LIN {X 0,Y 523.368,Z 555.346,A -85,B 0,C 180,E1 -4773.08,E2 -4773.08} C_VEL
LIN {X 0,Y 523.424,Z 552.407,A -85,B 0,C 180,E1 -4774.236,E2 -4774.236} C_VEL
LIN {X 0,Y 523.462,Z 548.426,A -85,B 0,C 180,E1 -4775.394,E2 -4775.394} C_VEL
LIN {X 0,Y 523.515,Z 542.323,A -85,B 0,C 180,E1 -4776.743,E2 -4776.743} C_VEL
LIN {X 0,Y 523.667,Z 535.613,A -85,B 0,C 180,E1 -4777.908,E2 -4777.908} C_VEL
LIN {X 0,Y 523.85,Z 527.313,A -85,B 0,C 180,E1 -4779.071,E2 -4779.071} C_VEL
LIN {X 0,Y 524.066,Z 518.806,A -85,B 0,C 180,E1 -4780.041,E2 -4780.041} C_VEL
LIN {X 0,Y 524.361,Z 508.295,A -85,B 0,C 180,E1 -4781.012,E2 -4781.012} C_VEL
LIN {X 0,Y 524.634,Z 497.983,A -85,B 0,C 180,E1 -4781.783,E2 -4781.783} C_VEL
LIN {X 0,Y 524.903,Z 486.499,A -85,B 0,C 180,E1 -4782.469,E2 -4782.469} C_VEL
LIN {X 0,Y 525.115,Z 474.788,A -85,B 0,C 180,E1 -4783.005,E2 -4783.005} C_VEL
LIN {X 0,Y 525.386,Z 461.299,A -85,B 0,C 180,E1 -4783.441,E2 -4783.441} C_VEL
LIN {X 0,Y 525.56,Z 447.895,A -85,B 0,C 180,E1 -4783.707,E2 -4783.707} C_VEL
LIN {X 0,Y 525.818,Z 355.734,A -85,B 0,C 180,E1 -4784.974,E2 -4784.974} C_VEL
LIN {X 0,Y 524.289,Z 345.618,A -85,B 0,C 180,E1 -4785.171,E2 -4785.171} C_VEL
LIN {X 0,Y 524.744,Z 323.595,A -85,B 0,C 180,E1 -4788.528,E2 -4788.528} C_VEL
LIN {X 0,Y 525.163,Z 305.11,A -85,B 0,C 180,E1 -4791.388,E2 -4791.388} C_VEL
LIN {X 0,Y 525.41,Z 293.296,A -85,B 0,C 180,E1 -4793.242,E2 -4793.242} C_VEL
LIN {X 0,Y 523.995,Z 285.213,A -85,B 0,C 180,E1 -4794.622,E2 -4794.622} C_VEL
LIN {X 0,Y 523.978,Z 285.217,A -85,B 0,C 180,E1 -4797.718,E2 -4797.718} C_VEL
LIN {X 0,Y 523.951,Z 285.214,A -85,B 0,C 180,E1 -4800.855,E2 -4800.855} C_VEL
LIN {X 0,Y 523.937,Z 285.217,A -85,B 0,C 180,E1 -4803.73,E2 -4803.73} C_VEL
LIN {X 0,Y 523.909,Z 285.228,A -85,B 0,C 180,E1 -4806.402,E2 -4806.402} C_VEL
LIN {X 0,Y 523.919,Z 285.218,A -85,B 0,C 180,E1 -4809.086,E2 -4809.086} C_VEL
LIN {X 0,Y 523.957,Z 285.216,A -85,B 0,C 180,E1 -4812.119,E2 -4812.119} C_VEL
LIN {X 0,Y 523.948,Z 285.215,A -85,B 0,C 180,E1 -4815.311,E2 -4815.311} C_VEL
LIN {X 0,Y 523.961,Z 285.221,A -85,B 0,C 180,E1 -4818.69,E2 -4818.69} C_VEL
LIN {X 0,Y 523.922,Z 285.223,A -85,B 0,C 180,E1 -4821.081,E2 -4821.081} C_VEL
LIN {X 0,Y 523.905,Z 285.219,A -85,B 0,C 180,E1 -4823.825,E2 -4823.825} C_VEL
LIN {X 0,Y 523.918,Z 285.221,A -85,B 0,C 180,E1 -4826.634,E2 -4826.634} C_VEL
LIN {X 0,Y 523.961,Z 285.218,A -85,B 0,C 180,E1 -4829.356,E2 -4829.356} C_VEL
LIN {X 0,Y 523.981,Z 285.209,A -85,B 0,C 180,E1 -4832.282,E2 -4832.282} C_VEL
LIN {X 0,Y 523.954,Z 285.214,A -85,B 0,C 180,E1 -4834.581,E2 -4834.581} C_VEL
LIN {X 0,Y 523.915,Z 285.224,A -85,B 0,C 180,E1 -4837.106,E2 -4837.106} C_VEL
LIN {X 0,Y 523.984,Z 285.212,A -85,B 0,C 180,E1 -4839.866,E2 -4839.866} C_VEL
LIN {X 0,Y 523.959,Z 285.213,A -85,B 0,C 180,E1 -4842.837,E2 -4842.837} C_VEL
LIN {X 0,Y 523.982,Z 285.213,A -85,B 0,C 180,E1 -4845.236,E2 -4845.236} C_VEL
LIN {X 0,Y 524.018,Z 285.206,A -85,B 0,C 180,E1 -4848.394,E2 -4848.394} C_VEL
LIN {X 0,Y 524.001,Z 285.212,A -85,B 0,C 180,E1 -4851.516,E2 -4851.516} C_VEL
LIN {X 0,Y 524.079,Z 285.198,A -85,B 0,C 180,E1 -4854.613,E2 -4854.613} C_VEL
LIN {X 0,Y 524.116,Z 285.197,A -85,B 0,C 180,E1 -4857.694,E2 -4857.694} C_VEL
LIN {X 0,Y 524.126,Z 285.193,A -85,B 0,C 180,E1 -4860.768,E2 -4860.768} C_VEL
LIN {X 0,Y 524.073,Z 285.198,A -85,B 0,C 180,E1 -4863.075,E2 -4863.075} C_VEL
LIN {X 0,Y 524.039,Z 285.21,A -85,B 0,C 180,E1 -4866.159,E2 -4866.159} C_VEL
LIN {X 0,Y 523.99,Z 285.208,A -85,B 0,C 180,E1 -4869.262,E2 -4869.262} C_VEL
LIN {X 0,Y 524.004,Z 285.207,A -85,B 0,C 180,E1 -4871.737,E2 -4871.737} C_VEL
LIN {X 0,Y 523.999,Z 285.21,A -85,B 0,C 180,E1 -4875.052,E2 -4875.052} C_VEL
LIN {X 0,Y 523.952,Z 285.214,A -85,B 0,C 180,E1 -4877.969,E2 -4877.969} C_VEL
LIN {X 0,Y 523.976,Z 285.214,A -85,B 0,C 180,E1 -4880.41,E2 -4880.41} C_VEL
LIN {X 0,Y 523.914,Z 285.228,A -85,B 0,C 180,E1 -4882.893,E2 -4882.893} C_VEL
LIN {X 0,Y 523.957,Z 285.215,A -85,B 0,C 180,E1 -4885.418,E2 -4885.418} C_VEL
LIN {X 0,Y 523.972,Z 285.21,A -85,B 0,C 180,E1 -4887.999,E2 -4887.999} C_VEL
LIN {X 0,Y 523.949,Z 285.219,A -85,B 0,C 180,E1 -4890.854,E2 -4890.854} C_VEL
LIN {X 0,Y 523.963,Z 285.214,A -85,B 0,C 180,E1 -4893.734,E2 -4893.734} C_VEL
LIN {X 0,Y 523.902,Z 285.219,A -85,B 0,C 180,E1 -4896.4,E2 -4896.4} C_VEL
LIN {X 0,Y 523.922,Z 285.222,A -85,B 0,C 180,E1 -4899.084,E2 -4899.084} C_VEL
LIN {X 0,Y 523.955,Z 285.214,A -85,B 0,C 180,E1 -4902.118,E2 -4902.118} C_VEL
LIN {X 0,Y 523.946,Z 285.219,A -85,B 0,C 180,E1 -4905.31,E2 -4905.31} C_VEL
LIN {X 0,Y 523.918,Z 285.218,A -85,B 0,C 180,E1 -4906.904,E2 -4906.904} C_VEL
LIN {X 0,Y 523.254,Z 285.308,A -85,B 0,C 180,E1 -4907.546,E2 -4907.546} C_VEL
LIN {X 0,Y 520.414,Z 285.662,A -85,B 0,C 180,E1 -4908.588,E2 -4908.588} C_VEL
LIN {X 0,Y 518.01,Z 285.961,A -85,B 0,C 180,E1 -4909.426,E2 -4909.426} C_VEL
LIN {X 0,Y 516.972,Z 286.088,A -85,B 0,C 180,E1 -4910.074,E2 -4910.074} C_VEL
LIN {X 0,Y 516.885,Z 286.096,A -85,B 0,C 180,E1 -4910.293,E2 -4910.293} C_VEL
LIN {X 0,Y 516.88,Z 286.096,A -85,B 0,C 180,E1 -4913.342,E2 -4913.342} C_VEL
LIN {X 0,Y 516.911,Z 286.097,A -85,B 0,C 180,E1 -4916.12,E2 -4916.12} C_VEL
LIN {X 0,Y 516.895,Z 286.092,A -85,B 0,C 180,E1 -4918.935,E2 -4918.935} C_VEL
LIN {X 0,Y 516.923,Z 286.091,A -85,B 0,C 180,E1 -4921.584,E2 -4921.584} C_VEL
LIN {X 0,Y 516.933,Z 286.098,A -85,B 0,C 180,E1 -4924.21,E2 -4924.21} C_VEL
LIN {X 0,Y 516.864,Z 286.099,A -85,B 0,C 180,E1 -4926.775,E2 -4926.775} C_VEL
LIN {X 0,Y 516.943,Z 286.087,A -85,B 0,C 180,E1 -4929.731,E2 -4929.731} C_VEL
LIN {X 0,Y 516.923,Z 286.097,A -85,B 0,C 180,E1 -4932.595,E2 -4932.595} C_VEL
LIN {X 0,Y 516.945,Z 286.089,A -85,B 0,C 180,E1 -4935.029,E2 -4935.029} C_VEL
LIN {X 0,Y 516.968,Z 286.086,A -85,B 0,C 180,E1 -4938.233,E2 -4938.233} C_VEL
LIN {X 0,Y 516.958,Z 286.088,A -85,B 0,C 180,E1 -4941.398,E2 -4941.398} C_VEL
LIN {X 0,Y 517.003,Z 286.083,A -85,B 0,C 180,E1 -4943.756,E2 -4943.756} C_VEL
LIN {X 0,Y 516.949,Z 286.257,A -85,B 0,C 180,E1 -4945.271,E2 -4945.271} C_VEL
LIN {X 0,Y 517.481,Z 291.535,A -85,B 0,C 180,E1 -4946.3,E2 -4946.3} C_VEL
LIN {X 0,Y 517.248,Z 305.925,A -85,B 0,C 180,E1 -4949.026,E2 -4949.026} C_VEL
LIN {X 0,Y 517.231,Z 309.396,A -85,B 0,C 180,E1 -4949.683,E2 -4949.683} C_VEL
LIN {X 0,Y 519.124,Z 320.066,A -85,B 0,C 180,E1 -4949.902,E2 -4949.902} C_VEL
LIN {X 0,Y 518.55,Z 416.495,A -85,B 0,C 180,E1 -4951.261,E2 -4951.261} C_VEL
LIN {X 0,Y 518.369,Z 430.247,A -85,B 0,C 180,E1 -4951.625,E2 -4951.625} C_VEL
LIN {X 0,Y 518.189,Z 442.011,A -85,B 0,C 180,E1 -4952.088,E2 -4952.088} C_VEL
LIN {X 0,Y 517.935,Z 453.991,A -85,B 0,C 180,E1 -4952.721,E2 -4952.721} C_VEL
LIN {X 0,Y 517.571,Z 465.423,A -85,B 0,C 180,E1 -4953.502,E2 -4953.502} C_VEL
LIN {X 0,Y 517.287,Z 475.712,A -85,B 0,C 180,E1 -4954.382,E2 -4954.382} C_VEL
LIN {X 0,Y 517.045,Z 484.149,A -85,B 0,C 180,E1 -4955.263,E2 -4955.263} C_VEL
LIN {X 0,Y 516.815,Z 491.954,A -85,B 0,C 180,E1 -4956.244,E2 -4956.244} C_VEL
LIN {X 0,Y 516.665,Z 499.581,A -85,B 0,C 180,E1 -4957.424,E2 -4957.424} C_VEL
LIN {X 0,Y 516.486,Z 505.737,A -85,B 0,C 180,E1 -4958.607,E2 -4958.607} C_VEL
LIN {X 0,Y 516.369,Z 510.631,A -85,B 0,C 180,E1 -4959.794,E2 -4959.794} C_VEL
LIN {X 0,Y 516.337,Z 514.4,A -85,B 0,C 180,E1 -4960.984,E2 -4960.984} C_VEL
LIN {X 0,Y 516.28,Z 516.352,A -85,B 0,C 180,E1 -4961.781,E2 -4961.781} C_VEL
LIN {X 0,Y 516.22,Z 517.869,A -85,B 0,C 180,E1 -4962.58,E2 -4962.58} C_VEL
LIN {X 0,Y 516.183,Z 518.924,A -85,B 0,C 180,E1 -4963.382,E2 -4963.382} C_VEL
LIN {X 0,Y 516.246,Z 519.808,A -85,B 0,C 180,E1 -4964.857,E2 -4964.857} C_VEL
LIN {X 0,Y 516.15,Z 519.646,A -85,B 0,C 180,E1 -4965.801,E2 -4965.801} C_VEL
LIN {X 0,Y 516.166,Z 519.025,A -85,B 0,C 180,E1 -4966.613,E2 -4966.613} C_VEL
LIN {X 0,Y 516.228,Z 517.656,A -85,B 0,C 180,E1 -4967.638,E2 -4967.638} C_VEL
LIN {X 0,Y 516.287,Z 514.52,A -85,B 0,C 180,E1 -4969.067,E2 -4969.067} C_VEL
LIN {X 0,Y 516.396,Z 510.398,A -85,B 0,C 180,E1 -4970.366,E2 -4970.366} C_VEL
LIN {X 0,Y 516.45,Z 505.433,A -85,B 0,C 180,E1 -4971.555,E2 -4971.555} C_VEL
LIN {X 0,Y 516.657,Z 498.795,A -85,B 0,C 180,E1 -4972.809,E2 -4972.809} C_VEL
LIN {X 0,Y 516.901,Z 490.288,A -85,B 0,C 180,E1 -4974.071,E2 -4974.071} C_VEL
LIN {X 0,Y 517.154,Z 481.46,A -85,B 0,C 180,E1 -4975.129,E2 -4975.129} C_VEL
LIN {X 0,Y 517.471,Z 471.556,A -85,B 0,C 180,E1 -4976.09,E2 -4976.09} C_VEL
LIN {X 0,Y 517.711,Z 460.662,A -85,B 0,C 180,E1 -4976.939,E2 -4976.939} C_VEL
LIN {X 0,Y 518.074,Z 448.787,A -85,B 0,C 180,E1 -4977.668,E2 -4977.668} C_VEL
LIN {X 0,Y 518.317,Z 437.639,A -85,B 0,C 180,E1 -4978.194,E2 -4978.194} C_VEL
LIN {X 0,Y 518.525,Z 425.119,A -85,B 0,C 180,E1 -4978.621,E2 -4978.621} C_VEL
LIN {X 0,Y 518.648,Z 412.955,A -85,B 0,C 180,E1 -4978.891,E2 -4978.891} C_VEL
LIN {X 0,Y 519.058,Z 319.441,A -85,B 0,C 180,E1 -4980.2,E2 -4980.2} C_VEL
LIN {X 0,Y 517.193,Z 309.171,A -85,B 0,C 180,E1 -4980.424,E2 -4980.424} C_VEL
LIN {X 0,Y 517.319,Z 292.962,A -85,B 0,C 180,E1 -4983.38,E2 -4983.38} C_VEL
LIN {X 0,Y 517.113,Z 287.483,A -85,B 0,C 180,E1 -4984.385,E2 -4984.385} C_VEL
LIN {X 0,Y 516.871,Z 286.105,A -85,B 0,C 180,E1 -4984.666,E2 -4984.666} C_VEL
LIN {X 0,Y 516.842,Z 286.103,A -85,B 0,C 180,E1 -4987.938,E2 -4987.938} C_VEL
LIN {X 0,Y 516.836,Z 286.104,A -85,B 0,C 180,E1 -4990.744,E2 -4990.744} C_VEL
LIN {X 0,Y 516.847,Z 286.102,A -85,B 0,C 180,E1 -4993.905,E2 -4993.905} C_VEL
LIN {X 0,Y 516.868,Z 286.095,A -85,B 0,C 180,E1 -4996.106,E2 -4996.106} C_VEL
LIN {X 0,Y 516.839,Z 286.106,A -85,B 0,C 180,E1 -4999.254,E2 -4999.254} C_VEL
LIN {X 0,Y 516.849,Z 286.103,A -85,B 0,C 180,E1 -5002.059,E2 -5002.059} C_VEL
LIN {X 0,Y 516.861,Z 286.094,A -85,B 0,C 180,E1 -5005.174,E2 -5005.174} C_VEL
LIN {X 0,Y 516.859,Z 286.102,A -85,B 0,C 180,E1 -5007.974,E2 -5007.974} C_VEL
LIN {X 0,Y 516.906,Z 286.092,A -85,B 0,C 180,E1 -5010.695,E2 -5010.695} C_VEL
LIN {X 0,Y 516.883,Z 286.104,A -85,B 0,C 180,E1 -5013.814,E2 -5013.814} C_VEL
LIN {X 0,Y 516.844,Z 286.1,A -85,B 0,C 180,E1 -5016.775,E2 -5016.775} C_VEL
LIN {X 0,Y 516.922,Z 286.092,A -85,B 0,C 180,E1 -5019.732,E2 -5019.732} C_VEL
LIN {X 0,Y 516.887,Z 286.094,A -85,B 0,C 180,E1 -5022.595,E2 -5022.595} C_VEL
LIN {X 0,Y 516.919,Z 286.09,A -85,B 0,C 180,E1 -5025.03,E2 -5025.03} C_VEL
LIN {X 0,Y 516.95,Z 286.091,A -85,B 0,C 180,E1 -5028.233,E2 -5028.233} C_VEL
LIN {X 0,Y 516.953,Z 286.086,A -85,B 0,C 180,E1 -5031.4,E2 -5031.4} C_VEL
LIN {X 0,Y 517.008,Z 286.086,A -85,B 0,C 180,E1 -5034.54,E2 -5034.54} C_VEL
LIN {X 0,Y 517.065,Z 286.07,A -85,B 0,C 180,E1 -5037.663,E2 -5037.663} C_VEL
LIN {X 0,Y 517.082,Z 286.074,A -85,B 0,C 180,E1 -5040.779,E2 -5040.779} C_VEL
LIN {X 0,Y 517.002,Z 286.077,A -85,B 0,C 180,E1 -5043.117,E2 -5043.117} C_VEL
LIN {X 0,Y 516.987,Z 286.085,A -85,B 0,C 180,E1 -5046.244,E2 -5046.244} C_VEL
LIN {X 0,Y 516.942,Z 286.086,A -85,B 0,C 180,E1 -5049.39,E2 -5049.39} C_VEL
LIN {X 0,Y 516.943,Z 286.086,A -85,B 0,C 180,E1 -5051.811,E2 -5051.811} C_VEL
LIN {X 0,Y 516.93,Z 286.094,A -85,B 0,C 180,E1 -5055.147,E2 -5055.147} C_VEL
LIN {X 0,Y 516.912,Z 286.09,A -85,B 0,C 180,E1 -5058.223,E2 -5058.223} C_VEL
LIN {X 0,Y 516.899,Z 286.096,A -85,B 0,C 180,E1 -5060.702,E2 -5060.702} C_VEL
LIN {X 0,Y 516.899,Z 286.09,A -85,B 0,C 180,E1 -5064.073,E2 -5064.073} C_VEL
LIN {X 0,Y 516.917,Z 286.093,A -85,B 0,C 180,E1 -5066.658,E2 -5066.658} C_VEL
LIN {X 0,Y 516.908,Z 286.096,A -85,B 0,C 180,E1 -5069.527,E2 -5069.527} C_VEL
LIN {X 0,Y 516.89,Z 286.092,A -85,B 0,C 180,E1 -5072.546,E2 -5072.546} C_VEL
LIN {X 0,Y 516.873,Z 286.104,A -85,B 0,C 180,E1 -5075.334,E2 -5075.334} C_VEL
LIN {X 0,Y 516.875,Z 286.098,A -85,B 0,C 180,E1 -5077.945,E2 -5077.945} C_VEL
LIN {X 0,Y 516.877,Z 286.097,A -85,B 0,C 180,E1 -5080.743,E2 -5080.743} C_VEL
LIN {X 0,Y 516.896,Z 286.093,A -85,B 0,C 180,E1 -5082.83,E2 -5082.83} C_VEL
LIN {X 0,Y 516.914,Z 286.092,A -85,B 0,C 180,E1 -5085.011,E2 -5085.011} C_VEL
LIN {X 0,Y 516.916,Z 286.092,A -85,B 0,C 180,E1 -5088.399,E2 -5088.399} C_VEL
LIN {X 0,Y 516.88,Z 286.097,A -85,B 0,C 180,E1 -5091.286,E2 -5091.286} C_VEL
LIN {X 0,Y 516.883,Z 286.1,A -85,B 0,C 180,E1 -5094.223,E2 -5094.223} C_VEL
LIN {X 0,Y 516.89,Z 286.094,A -85,B 0,C 180,E1 -5097.055,E2 -5097.055} C_VEL
LIN {X 0,Y 516.888,Z 286.102,A -85,B 0,C 180,E1 -5099.798,E2 -5099.798} C_VEL
LIN {X 0,Y 516.926,Z 286.096,A -85,B 0,C 180,E1 -5102.469,E2 -5102.469} C_VEL
LIN {X 0,Y 516.965,Z 286.235,A -85,B 0,C 180,E1 -5105.338,E2 -5105.338} C_VEL
LIN {X 0,Y 518.468,Z 295.266,A -85,B 0,C 180,E1 -5106.854,E2 -5106.854} C_VEL
LIN {X 0,Y 517.946,Z 315.173,A -85,B 0,C 180,E1 -5109.979,E2 -5109.979} C_VEL
LIN {X 0,Y 517.475,Z 333.55,A -85,B 0,C 180,E1 -5112.82,E2 -5112.82} C_VEL
LIN {X 0,Y 517.256,Z 345.372,A -85,B 0,C 180,E1 -5114.631,E2 -5114.631} C_VEL
LIN {X 0,Y 519.048,Z 357.786,A -85,B 0,C 180,E1 -5114.86,E2 -5114.86} C_VEL
LIN {X 0,Y 518.578,Z 453.593,A -85,B 0,C 180,E1 -5116.207,E2 -5116.207} C_VEL
LIN {X 0,Y 518.356,Z 466.931,A -85,B 0,C 180,E1 -5116.551,E2 -5116.551} C_VEL
LIN {X 0,Y 518.057,Z 480.264,A -85,B 0,C 180,E1 -5117.067,E2 -5117.067} C_VEL
LIN {X 0,Y 517.82,Z 492.824,A -85,B 0,C 180,E1 -5117.744,E2 -5117.744} C_VEL
LIN {X 0,Y 517.545,Z 503.086,A -85,B 0,C 180,E1 -5118.447,E2 -5118.447} C_VEL
LIN {X 0,Y 517.216,Z 513.557,A -85,B 0,C 180,E1 -5119.332,E2 -5119.332} C_VEL
LIN {X 0,Y 516.957,Z 522.12,A -85,B 0,C 180,E1 -5120.217,E2 -5120.217} C_VEL
LIN {X 0,Y 516.709,Z 530.021,A -85,B 0,C 180,E1 -5121.2,E2 -5121.2} C_VEL
LIN {X 0,Y 516.543,Z 537.74,A -85,B 0,C 180,E1 -5122.378,E2 -5122.378} C_VEL
LIN {X 0,Y 516.4,Z 544.856,A -85,B 0,C 180,E1 -5123.751,E2 -5123.751} C_VEL
LIN {X 0,Y 516.313,Z 549.59,A -85,B 0,C 180,E1 -5124.925,E2 -5124.925} C_VEL
LIN {X 0,Y 516.352,Z 553.211,A -85,B 0,C 180,E1 -5126.099,E2 -5126.099} C_VEL
LIN {X 0,Y 516.282,Z 555.075,A -85,B 0,C 180,E1 -5126.88,E2 -5126.88} C_VEL
LIN {X 0,Y 516.26,Z 556.474,A -85,B 0,C 180,E1 -5127.661,E2 -5127.661} C_VEL
LIN {X 0,Y 516.16,Z 558.08,A -85,B 0,C 180,E1 -5129.221,E2 -5129.221} C_VEL
LIN {X 0,Y 516.158,Z 558.297,A -85,B 0,C 180,E1 -5130.001,E2 -5130.001} C_VEL
LIN {X 0,Y 516.192,Z 557.474,A -85,B 0,C 180,E1 -5131.562,E2 -5131.562} C_VEL
LIN {X 0,Y 516.261,Z 556.48,A -85,B 0,C 180,E1 -5132.342,E2 -5132.342} C_VEL
LIN {X 0,Y 516.283,Z 555.083,A -85,B 0,C 180,E1 -5133.122,E2 -5133.122} C_VEL
LIN {X 0,Y 516.312,Z 552.142,A -85,B 0,C 180,E1 -5134.295,E2 -5134.295} C_VEL
LIN {X 0,Y 516.376,Z 548.162,A -85,B 0,C 180,E1 -5135.468,E2 -5135.468} C_VEL
LIN {X 0,Y 516.423,Z 542.94,A -85,B 0,C 180,E1 -5136.664,E2 -5136.664} C_VEL
LIN {X 0,Y 516.582,Z 536.586,A -85,B 0,C 180,E1 -5137.82,E2 -5137.82} C_VEL
LIN {X 0,Y 516.77,Z 528.539,A -85,B 0,C 180,E1 -5138.999,E2 -5138.999} C_VEL
LIN {X 0,Y 516.987,Z 520.341,A -85,B 0,C 180,E1 -5139.982,E2 -5139.982} C_VEL
LIN {X 0,Y 517.272,Z 510.344,A -85,B 0,C 180,E1 -5140.966,E2 -5140.966} C_VEL
LIN {X 0,Y 517.627,Z 500.483,A -85,B 0,C 180,E1 -5141.752,E2 -5141.752} C_VEL
LIN {X 0,Y 517.854,Z 489.323,A -85,B 0,C 180,E1 -5142.468,E2 -5142.468} C_VEL
LIN {X 0,Y 518.145,Z 476.865,A -85,B 0,C 180,E1 -5143.083,E2 -5143.083} C_VEL
LIN {X 0,Y 518.402,Z 463.75,A -85,B 0,C 180,E1 -5143.55,E2 -5143.55} C_VEL
LIN {X 0,Y 518.643,Z 450.635,A -85,B 0,C 180,E1 -5143.844,E2 -5143.844} C_VEL
LIN {X 0,Y 519.049,Z 357.444,A -85,B 0,C 180,E1 -5145.146,E2 -5145.146} C_VEL
LIN {X 0,Y 517.27,Z 345.411,A -85,B 0,C 180,E1 -5145.373,E2 -5145.373} C_VEL
LIN {X 0,Y 517.751,Z 324.521,A -85,B 0,C 180,E1 -5148.603,E2 -5148.603} C_VEL
LIN {X 0,Y 518.201,Z 306.177,A -85,B 0,C 180,E1 -5151.481,E2 -5151.481} C_VEL
LIN {X 0,Y 518.448,Z 294.349,A -85,B 0,C 180,E1 -5153.361,E2 -5153.361} C_VEL
LIN {X 0,Y 516.941,Z 286.092,A -85,B 0,C 180,E1 -5154.783,E2 -5154.783} C_VEL
LIN {X 0,Y 516.928,Z 286.094,A -85,B 0,C 180,E1 -5157.534,E2 -5157.534} C_VEL
LIN {X 0,Y 516.898,Z 286.102,A -85,B 0,C 180,E1 -5160.204,E2 -5160.204} C_VEL
LIN {X 0,Y 516.887,Z 286.094,A -85,B 0,C 180,E1 -5162.948,E2 -5162.948} C_VEL
LIN {X 0,Y 516.876,Z 286.097,A -85,B 0,C 180,E1 -5165.781,E2 -5165.781} C_VEL
LIN {X 0,Y 516.883,Z 286.099,A -85,B 0,C 180,E1 -5168.717,E2 -5168.717} C_VEL
LIN {X 0,Y 516.917,Z 286.09,A -85,B 0,C 180,E1 -5171.776,E2 -5171.776} C_VEL
LIN {X 0,Y 516.901,Z 286.095,A -85,B 0,C 180,E1 -5175.007,E2 -5175.007} C_VEL
LIN {X 0,Y 516.919,Z 286.094,A -85,B 0,C 180,E1 -5178.399,E2 -5178.399} C_VEL
LIN {X 0,Y 516.885,Z 286.096,A -85,B 0,C 180,E1 -5181.284,E2 -5181.284} C_VEL
LIN {X 0,Y 516.876,Z 286.095,A -85,B 0,C 180,E1 -5184.22,E2 -5184.22} C_VEL
LIN {X 0,Y 516.886,Z 286.103,A -85,B 0,C 180,E1 -5187.052,E2 -5187.052} C_VEL
LIN {X 0,Y 516.898,Z 286.093,A -85,B 0,C 180,E1 -5189.796,E2 -5189.796} C_VEL
LIN {X 0,Y 516.93,Z 286.088,A -85,B 0,C 180,E1 -5192.467,E2 -5192.467} C_VEL
LIN {X 0,Y 516.911,Z 286.097,A -85,B 0,C 180,E1 -5195.072,E2 -5195.072} C_VEL
LIN {X 0,Y 516.89,Z 286.093,A -85,B 0,C 180,E1 -5198.462,E2 -5198.462} C_VEL
LIN {X 0,Y 516.904,Z 286.093,A -85,B 0,C 180,E1 -5200.955,E2 -5200.955} C_VEL
LIN {X 0,Y 516.909,Z 286.098,A -85,B 0,C 180,E1 -5203.41,E2 -5203.41} C_VEL
LIN {X 0,Y 516.897,Z 286.099,A -85,B 0,C 180,E1 -5205.834,E2 -5205.834} C_VEL
LIN {X 0,Y 516.955,Z 286.086,A -85,B 0,C 180,E1 -5209.028,E2 -5209.028} C_VEL
LIN {X 0,Y 516.982,Z 286.086,A -85,B 0,C 180,E1 -5212.187,E2 -5212.187} C_VEL
LIN {X 0,Y 517.026,Z 286.077,A -85,B 0,C 180,E1 -5214.54,E2 -5214.54} C_VEL
LIN {X 0,Y 517.088,Z 286.072,A -85,B 0,C 180,E1 -5217.663,E2 -5217.663} C_VEL
LIN {X 0,Y 517.096,Z 286.068,A -85,B 0,C 180,E1 -5220.779,E2 -5220.779} C_VEL
LIN {X 0,Y 517.014,Z 286.077,A -85,B 0,C 180,E1 -5223.117,E2 -5223.117} C_VEL
LIN {X 0,Y 517.005,Z 286.088,A -85,B 0,C 180,E1 -5226.243,E2 -5226.243} C_VEL
LIN {X 0,Y 516.946,Z 286.086,A -85,B 0,C 180,E1 -5229.389,E2 -5229.389} C_VEL
LIN {X 0,Y 516.957,Z 286.085,A -85,B 0,C 180,E1 -5231.807,E2 -5231.807} C_VEL
LIN {X 0,Y 516.952,Z 286.087,A -85,B 0,C 180,E1 -5235.147,E2 -5235.147} C_VEL
LIN {X 0,Y 516.92,Z 286.092,A -85,B 0,C 180,E1 -5238.222,E2 -5238.222} C_VEL
LIN {X 0,Y 516.917,Z 286.098,A -85,B 0,C 180,E1 -5240.701,E2 -5240.701} C_VEL
LIN {X 0,Y 516.906,Z 286.091,A -85,B 0,C 180,E1 -5244.072,E2 -5244.072} C_VEL
LIN {X 0,Y 516.929,Z 286.093,A -85,B 0,C 180,E1 -5246.657,E2 -5246.657} C_VEL
LIN {X 0,Y 516.915,Z 286.093,A -85,B 0,C 180,E1 -5249.523,E2 -5249.523} C_VEL
LIN {X 0,Y 516.9,Z 286.093,A -85,B 0,C 180,E1 -5252.543,E2 -5252.543} C_VEL
LIN {X 0,Y 516.868,Z 286.105,A -85,B 0,C 180,E1 -5255.329,E2 -5255.329} C_VEL
LIN {X 0,Y 516.882,Z 286.095,A -85,B 0,C 180,E1 -5257.942,E2 -5257.942} C_VEL
LIN {X 0,Y 516.887,Z 286.094,A -85,B 0,C 180,E1 -5260.741,E2 -5260.741} C_VEL
LIN {X 0,Y 516.886,Z 286.094,A -85,B 0,C 180,E1 -5262.831,E2 -5262.831} C_VEL
LIN {X 0,Y 516.899,Z 286.094,A -85,B 0,C 180,E1 -5265.006,E2 -5265.006} C_VEL
LIN {X 0,Y 516.917,Z 286.09,A -85,B 0,C 180,E1 -5268.398,E2 -5268.398} C_VEL
LIN {X 0,Y 516.885,Z 286.096,A -85,B 0,C 180,E1 -5270.293,E2 -5270.293} C_VEL
LIN {X 0,Y 516.213,Z 286.178,A -85,B 0,C 180,E1 -5270.944,E2 -5270.944} C_VEL
LIN {X 0,Y 513.366,Z 286.539,A -85,B 0,C 180,E1 -5271.999,E2 -5271.999} C_VEL
LIN {X 0,Y 510.957,Z 286.842,A -85,B 0,C 180,E1 -5272.849,E2 -5272.849} C_VEL
LIN {X 0,Y 509.914,Z 286.969,A -85,B 0,C 180,E1 -5273.506,E2 -5273.506} C_VEL
LIN {X 0,Y 509.824,Z 286.978,A -85,B 0,C 180,E1 -5273.728,E2 -5273.728} C_VEL
LIN {X 0,Y 509.862,Z 286.97,A -85,B 0,C 180,E1 -5276.538,E2 -5276.538} C_VEL
LIN {X 0,Y 509.849,Z 286.971,A -85,B 0,C 180,E1 -5279.334,E2 -5279.334} C_VEL
LIN {X 0,Y 509.898,Z 286.972,A -85,B 0,C 180,E1 -5282.054,E2 -5282.054} C_VEL
LIN {X 0,Y 509.844,Z 286.973,A -85,B 0,C 180,E1 -5284.701,E2 -5284.701} C_VEL
LIN {X 0,Y 509.83,Z 286.973,A -85,B 0,C 180,E1 -5287.457,E2 -5287.457} C_VEL
LIN {X 0,Y 509.92,Z 286.963,A -85,B 0,C 180,E1 -5289.844,E2 -5289.844} C_VEL
LIN {X 0,Y 509.882,Z 286.967,A -85,B 0,C 180,E1 -5293.174,E2 -5293.174} C_VEL
LIN {X 0,Y 509.865,Z 286.968,A -85,B 0,C 180,E1 -5295.633,E2 -5295.633} C_VEL
LIN {X 0,Y 509.915,Z 286.969,A -85,B 0,C 180,E1 -5298.874,E2 -5298.874} C_VEL
LIN {X 0,Y 509.923,Z 286.964,A -85,B 0,C 180,E1 -5302.077,E2 -5302.077} C_VEL
LIN {X 0,Y 509.933,Z 286.97,A -85,B 0,C 180,E1 -5305.057,E2 -5305.057} C_VEL
LIN {X 0,Y 509.997,Z 287.671,A -85,B 0,C 180,E1 -5305.256,E2 -5305.256} C_VEL
LIN {X 0,Y 510.495,Z 292.734,A -85,B 0,C 180,E1 -5306.249,E2 -5306.249} C_VEL
LIN {X 0,Y 510.25,Z 307.211,A -85,B 0,C 180,E1 -5309.012,E2 -5309.012} C_VEL
LIN {X 0,Y 510.255,Z 309.888,A -85,B 0,C 180,E1 -5309.481,E2 -5309.481} C_VEL
LIN {X 0,Y 512.286,Z 320.969,A -85,B 0,C 180,E1 -5309.704,E2 -5309.704} C_VEL
LIN {X 0,Y 511.688,Z 417.1,A -85,B 0,C 180,E1 -5311.081,E2 -5311.081} C_VEL
LIN {X 0,Y 511.461,Z 430.768,A -85,B 0,C 180,E1 -5311.451,E2 -5311.451} C_VEL
LIN {X 0,Y 511.281,Z 443.5,A -85,B 0,C 180,E1 -5311.968,E2 -5311.968} C_VEL
LIN {X 0,Y 510.907,Z 455.971,A -85,B 0,C 180,E1 -5312.66,E2 -5312.66} C_VEL
LIN {X 0,Y 510.593,Z 467.063,A -85,B 0,C 180,E1 -5313.451,E2 -5313.451} C_VEL
LIN {X 0,Y 510.278,Z 477.089,A -85,B 0,C 180,E1 -5314.343,E2 -5314.343} C_VEL
LIN {X 0,Y 509.964,Z 486.151,A -85,B 0,C 180,E1 -5315.336,E2 -5315.336} C_VEL
LIN {X 0,Y 509.739,Z 494.727,A -85,B 0,C 180,E1 -5316.492,E2 -5316.492} C_VEL
LIN {X 0,Y 509.554,Z 502.118,A -85,B 0,C 180,E1 -5317.727,E2 -5317.727} C_VEL
LIN {X 0,Y 509.411,Z 506.945,A -85,B 0,C 180,E1 -5318.728,E2 -5318.728} C_VEL
LIN {X 0,Y 509.285,Z 511.643,A -85,B 0,C 180,E1 -5319.932,E2 -5319.932} C_VEL
LIN {X 0,Y 509.267,Z 515.224,A -85,B 0,C 180,E1 -5321.138,E2 -5321.138} C_VEL
LIN {X 0,Y 509.169,Z 517.061,A -85,B 0,C 180,E1 -5321.948,E2 -5321.948} C_VEL
LIN {X 0,Y 509.13,Z 518.431,A -85,B 0,C 180,E1 -5322.758,E2 -5322.758} C_VEL
LIN {X 0,Y 509.092,Z 519.401,A -85,B 0,C 180,E1 -5323.572,E2 -5323.572} C_VEL
LIN {X 0,Y 509.147,Z 520.088,A -85,B 0,C 180,E1 -5324.93,E2 -5324.93} C_VEL
LIN {X 0,Y 509.051,Z 519.781,A -85,B 0,C 180,E1 -5326.027,E2 -5326.027} C_VEL
LIN {X 0,Y 509.08,Z 519.074,A -85,B 0,C 180,E1 -5326.851,E2 -5326.851} C_VEL
LIN {X 0,Y 509.137,Z 517.805,A -85,B 0,C 180,E1 -5327.739,E2 -5327.739} C_VEL
LIN {X 0,Y 509.204,Z 515.314,A -85,B 0,C 180,E1 -5328.924,E2 -5328.924} C_VEL
LIN {X 0,Y 509.302,Z 511.432,A -85,B 0,C 180,E1 -5330.224,E2 -5330.224} C_VEL
LIN {X 0,Y 509.377,Z 506.606,A -85,B 0,C 180,E1 -5331.445,E2 -5331.445} C_VEL
LIN {X 0,Y 509.608,Z 500.201,A -85,B 0,C 180,E1 -5332.713,E2 -5332.713} C_VEL
LIN {X 0,Y 509.781,Z 493.538,A -85,B 0,C 180,E1 -5333.78,E2 -5333.78} C_VEL
LIN {X 0,Y 510.026,Z 485.245,A -85,B 0,C 180,E1 -5334.87,E2 -5334.87} C_VEL
LIN {X 0,Y 510.348,Z 475.264,A -85,B 0,C 180,E1 -5335.926,E2 -5335.926} C_VEL
LIN {X 0,Y 510.693,Z 464.226,A -85,B 0,C 180,E1 -5336.863,E2 -5336.863} C_VEL
LIN {X 0,Y 511.065,Z 452.398,A -85,B 0,C 180,E1 -5337.652,E2 -5337.652} C_VEL
LIN {X 0,Y 511.337,Z 440.688,A -85,B 0,C 180,E1 -5338.252,E2 -5338.252} C_VEL
LIN {X 0,Y 511.614,Z 427.831,A -85,B 0,C 180,E1 -5338.735,E2 -5338.735} C_VEL
LIN {X 0,Y 511.748,Z 415.811,A -85,B 0,C 180,E1 -5339.036,E2 -5339.036} C_VEL
LIN {X 0,Y 512.189,Z 320.063,A -85,B 0,C 180,E1 -5340.403,E2 -5340.403} C_VEL
LIN {X 0,Y 510.208,Z 309.39,A -85,B 0,C 180,E1 -5340.64,E2 -5340.64} C_VEL
LIN {X 0,Y 510.38,Z 292.926,A -85,B 0,C 180,E1 -5343.657,E2 -5343.657} C_VEL
LIN {X 0,Y 509.868,Z 287.278,A -85,B 0,C 180,E1 -5344.71,E2 -5344.71} C_VEL
LIN {X 0,Y 509.828,Z 286.983,A -85,B 0,C 180,E1 -5344.893,E2 -5344.893} C_VEL
LIN {X 0,Y 509.798,Z 286.98,A -85,B 0,C 180,E1 -5348.341,E2 -5348.341} C_VEL
LIN {X 0,Y 509.789,Z 286.986,A -85,B 0,C 180,E1 -5351.43,E2 -5351.43} C_VEL
LIN {X 0,Y 509.822,Z 286.976,A -85,B 0,C 180,E1 -5354.669,E2 -5354.669} C_VEL
LIN {X 0,Y 509.789,Z 286.987,A -85,B 0,C 180,E1 -5357.506,E2 -5357.506} C_VEL
LIN {X 0,Y 509.818,Z 286.976,A -85,B 0,C 180,E1 -5360.645,E2 -5360.645} C_VEL
LIN {X 0,Y 509.784,Z 286.982,A -85,B 0,C 180,E1 -5363.644,E2 -5363.644} C_VEL
LIN {X 0,Y 509.827,Z 286.974,A -85,B 0,C 180,E1 -5366.537,E2 -5366.537} C_VEL
LIN {X 0,Y 509.831,Z 286.975,A -85,B 0,C 180,E1 -5369.333,E2 -5369.333} C_VEL
LIN {X 0,Y 509.831,Z 286.979,A -85,B 0,C 180,E1 -5372.051,E2 -5372.051} C_VEL
LIN {X 0,Y 509.803,Z 286.975,A -85,B 0,C 180,E1 -5374.7,E2 -5374.7} C_VEL
LIN {X 0,Y 509.811,Z 286.978,A -85,B 0,C 180,E1 -5377.458,E2 -5377.458} C_VEL
LIN {X 0,Y 509.9,Z 286.968,A -85,B 0,C 180,E1 -5379.844,E2 -5379.844} C_VEL
LIN {X 0,Y 509.85,Z 286.968,A -85,B 0,C 180,E1 -5383.174,E2 -5383.174} C_VEL
LIN {X 0,Y 509.841,Z 286.974,A -85,B 0,C 180,E1 -5385.634,E2 -5385.634} C_VEL
LIN {X 0,Y 509.897,Z 286.965,A -85,B 0,C 180,E1 -5388.874,E2 -5388.874} C_VEL
LIN {X 0,Y 509.936,Z 286.966,A -85,B 0,C 180,E1 -5392.078,E2 -5392.078} C_VEL
LIN {X 0,Y 509.958,Z 286.965,A -85,B 0,C 180,E1 -5394.464,E2 -5394.464} C_VEL
LIN {X 0,Y 510.036,Z 286.945,A -85,B 0,C 180,E1 -5397.631,E2 -5397.631} C_VEL
LIN {X 0,Y 510.052,Z 286.95,A -85,B 0,C 180,E1 -5400.79,E2 -5400.79} C_VEL
LIN {X 0,Y 509.943,Z 286.956,A -85,B 0,C 180,E1 -5403.16,E2 -5403.16} C_VEL
LIN {X 0,Y 509.938,Z 286.964,A -85,B 0,C 180,E1 -5406.33,E2 -5406.33} C_VEL
LIN {X 0,Y 509.903,Z 286.968,A -85,B 0,C 180,E1 -5408.721,E2 -5408.721} C_VEL
LIN {X 0,Y 509.891,Z 286.965,A -85,B 0,C 180,E1 -5411.932,E2 -5411.932} C_VEL
LIN {X 0,Y 509.88,Z 286.971,A -85,B 0,C 180,E1 -5415.242,E2 -5415.242} C_VEL
LIN {X 0,Y 509.875,Z 286.966,A -85,B 0,C 180,E1 -5418.002,E2 -5418.002} C_VEL
LIN {X 0,Y 509.837,Z 286.981,A -85,B 0,C 180,E1 -5421.002,E2 -5421.002} C_VEL
LIN {X 0,Y 509.824,Z 286.974,A -85,B 0,C 180,E1 -5423.564,E2 -5423.564} C_VEL
LIN {X 0,Y 509.902,Z 286.965,A -85,B 0,C 180,E1 -5426.38,E2 -5426.38} C_VEL
LIN {X 0,Y 509.87,Z 286.969,A -85,B 0,C 180,E1 -5428.845,E2 -5428.845} C_VEL
LIN {X 0,Y 509.816,Z 286.977,A -85,B 0,C 180,E1 -5431.591,E2 -5431.591} C_VEL
LIN {X 0,Y 509.844,Z 286.972,A -85,B 0,C 180,E1 -5434.414,E2 -5434.414} C_VEL
LIN {X 0,Y 509.812,Z 286.984,A -85,B 0,C 180,E1 -5437.341,E2 -5437.341} C_VEL
LIN {X 0,Y 509.83,Z 286.974,A -85,B 0,C 180,E1 -5440.383,E2 -5440.383} C_VEL
LIN {X 0,Y 509.831,Z 286.975,A -85,B 0,C 180,E1 -5443.066,E2 -5443.066} C_VEL
LIN {X 0,Y 509.823,Z 286.976,A -85,B 0,C 180,E1 -5445.794,E2 -5445.794} C_VEL
LIN {X 0,Y 509.859,Z 286.97,A -85,B 0,C 180,E1 -5448.577,E2 -5448.577} C_VEL
LIN {X 0,Y 509.846,Z 286.981,A -85,B 0,C 180,E1 -5451.788,E2 -5451.788} C_VEL
LIN {X 0,Y 509.838,Z 286.975,A -85,B 0,C 180,E1 -5454.624,E2 -5454.624} C_VEL
LIN {X 0,Y 509.856,Z 286.974,A -85,B 0,C 180,E1 -5457.482,E2 -5457.482} C_VEL
LIN {X 0,Y 509.855,Z 286.976,A -85,B 0,C 180,E1 -5460.275,E2 -5460.275} C_VEL
LIN {X 0,Y 509.883,Z 286.97,A -85,B 0,C 180,E1 -5462.946,E2 -5462.946} C_VEL
LIN {X 0,Y 509.92,Z 287.117,A -85,B 0,C 180,E1 -5465.158,E2 -5465.158} C_VEL
LIN {X 0,Y 511.369,Z 295.005,A -85,B 0,C 180,E1 -5466.513,E2 -5466.513} C_VEL
LIN {X 0,Y 511.222,Z 305.576,A -85,B 0,C 180,E1 -5468.213,E2 -5468.213} C_VEL
LIN {X 0,Y 510.739,Z 325.363,A -85,B 0,C 180,E1 -5471.343,E2 -5471.343} C_VEL
LIN {X 0,Y 510.263,Z 345.329,A -85,B 0,C 180,E1 -5474.419,E2 -5474.419} C_VEL
LIN {X 0,Y 512.208,Z 358.446,A -85,B 0,C 180,E1 -5474.666,E2 -5474.666} C_VEL
LIN {X 0,Y 511.698,Z 453.274,A -85,B 0,C 180,E1 -5476.018,E2 -5476.018} C_VEL
LIN {X 0,Y 511.453,Z 466.628,A -85,B 0,C 180,E1 -5476.366,E2 -5476.366} C_VEL
LIN {X 0,Y 511.137,Z 479.969,A -85,B 0,C 180,E1 -5476.888,E2 -5476.888} C_VEL
LIN {X 0,Y 510.891,Z 491.473,A -85,B 0,C 180,E1 -5477.508,E2 -5477.508} C_VEL
LIN {X 0,Y 510.548,Z 502.801,A -85,B 0,C 180,E1 -5478.286,E2 -5478.286} C_VEL
LIN {X 0,Y 510.221,Z 513.276,A -85,B 0,C 180,E1 -5479.184,E2 -5479.184} C_VEL
LIN {X 0,Y 509.921,Z 521.84,A -85,B 0,C 180,E1 -5480.081,E2 -5480.081} C_VEL
LIN {X 0,Y 509.664,Z 529.744,A -85,B 0,C 180,E1 -5481.077,E2 -5481.077} C_VEL
LIN {X 0,Y 509.478,Z 537.466,A -85,B 0,C 180,E1 -5482.272,E2 -5482.272} C_VEL
LIN {X 0,Y 509.316,Z 543.727,A -85,B 0,C 180,E1 -5483.477,E2 -5483.477} C_VEL
LIN {X 0,Y 509.243,Z 549.321,A -85,B 0,C 180,E1 -5484.855,E2 -5484.855} C_VEL
LIN {X 0,Y 509.245,Z 552.942,A -85,B 0,C 180,E1 -5486.044,E2 -5486.044} C_VEL
LIN {X 0,Y 509.2,Z 554.809,A -85,B 0,C 180,E1 -5486.836,E2 -5486.836} C_VEL
LIN {X 0,Y 509.189,Z 556.209,A -85,B 0,C 180,E1 -5487.628,E2 -5487.628} C_VEL
LIN {X 0,Y 509.073,Z 557.815,A -85,B 0,C 180,E1 -5489.21,E2 -5489.21} C_VEL
LIN {X 0,Y 509.069,Z 558.033,A -85,B 0,C 180,E1 -5490.001,E2 -5490.001} C_VEL
LIN {X 0,Y 509.112,Z 557.211,A -85,B 0,C 180,E1 -5491.583,E2 -5491.583} C_VEL
LIN {X 0,Y 509.189,Z 556.218,A -85,B 0,C 180,E1 -5492.374,E2 -5492.374} C_VEL
LIN {X 0,Y 509.201,Z 554.819,A -85,B 0,C 180,E1 -5493.166,E2 -5493.166} C_VEL
LIN {X 0,Y 509.204,Z 551.878,A -85,B 0,C 180,E1 -5494.355,E2 -5494.355} C_VEL
LIN {X 0,Y 509.293,Z 547.897,A -85,B 0,C 180,E1 -5495.544,E2 -5495.544} C_VEL
LIN {X 0,Y 509.401,Z 541.874,A -85,B 0,C 180,E1 -5496.915,E2 -5496.915} C_VEL
LIN {X 0,Y 509.545,Z 535.08,A -85,B 0,C 180,E1 -5498.129,E2 -5498.129} C_VEL
LIN {X 0,Y 509.757,Z 526.777,A -85,B 0,C 180,E1 -5499.324,E2 -5499.324} C_VEL
LIN {X 0,Y 509.996,Z 518.265,A -85,B 0,C 180,E1 -5500.321,E2 -5500.321} C_VEL
LIN {X 0,Y 510.391,Z 507.752,A -85,B 0,C 180,E1 -5501.317,E2 -5501.317} C_VEL
LIN {X 0,Y 510.671,Z 497.432,A -85,B 0,C 180,E1 -5502.11,E2 -5502.11} C_VEL
LIN {X 0,Y 511.007,Z 485.943,A -85,B 0,C 180,E1 -5502.814,E2 -5502.814} C_VEL
LIN {X 0,Y 511.248,Z 474.217,A -85,B 0,C 180,E1 -5503.364,E2 -5503.364} C_VEL
LIN {X 0,Y 511.6,Z 460.712,A -85,B 0,C 180,E1 -5503.81,E2 -5503.81} C_VEL
LIN {X 0,Y 511.786,Z 447.247,A -85,B 0,C 180,E1 -5504.084,E2 -5504.084} C_VEL
LIN {X 0,Y 512.112,Z 357.167,A -85,B 0,C 180,E1 -5505.357,E2 -5505.357} C_VEL
LIN {X 0,Y 510.246,Z 345.168,A -85,B 0,C 180,E1 -5505.587,E2 -5505.587} C_VEL
LIN {X 0,Y 510.749,Z 325.583,A -85,B 0,C 180,E1 -5508.659,E2 -5508.659} C_VEL
LIN {X 0,Y 511.249,Z 307.214,A -85,B 0,C 180,E1 -5511.576,E2 -5511.576} C_VEL
LIN {X 0,Y 511.465,Z 295.38,A -85,B 0,C 180,E1 -5513.485,E2 -5513.485} C_VEL
LIN {X 0,Y 509.909,Z 286.968,A -85,B 0,C 180,E1 -5514.955,E2 -5514.955} C_VEL
LIN {X 0,Y 509.89,Z 286.974,A -85,B 0,C 180,E1 -5517.947,E2 -5517.947} C_VEL
LIN {X 0,Y 509.851,Z 286.972,A -85,B 0,C 180,E1 -5520.666,E2 -5520.666} C_VEL
LIN {X 0,Y 509.848,Z 286.97,A -85,B 0,C 180,E1 -5523.463,E2 -5523.463} C_VEL
LIN {X 0,Y 509.83,Z 286.982,A -85,B 0,C 180,E1 -5526.354,E2 -5526.354} C_VEL
LIN {X 0,Y 509.84,Z 286.971,A -85,B 0,C 180,E1 -5529.354,E2 -5529.354} C_VEL
LIN {X 0,Y 509.839,Z 286.98,A -85,B 0,C 180,E1 -5532.49,E2 -5532.49} C_VEL
LIN {X 0,Y 509.845,Z 286.971,A -85,B 0,C 180,E1 -5535.33,E2 -5535.33} C_VEL
LIN {X 0,Y 509.861,Z 286.976,A -85,B 0,C 180,E1 -5538.575,E2 -5538.575} C_VEL
LIN {X 0,Y 509.856,Z 286.969,A -85,B 0,C 180,E1 -5541.787,E2 -5541.787} C_VEL
LIN {X 0,Y 509.834,Z 286.976,A -85,B 0,C 180,E1 -5544.622,E2 -5544.622} C_VEL
LIN {X 0,Y 509.865,Z 286.971,A -85,B 0,C 180,E1 -5547.481,E2 -5547.481} C_VEL
LIN {X 0,Y 509.864,Z 286.968,A -85,B 0,C 180,E1 -5550.274,E2 -5550.274} C_VEL
LIN {X 0,Y 509.888,Z 286.97,A -85,B 0,C 180,E1 -5552.944,E2 -5552.944} C_VEL
LIN {X 0,Y 509.867,Z 286.973,A -85,B 0,C 180,E1 -5555.574,E2 -5555.574} C_VEL
LIN {X 0,Y 509.855,Z 286.973,A -85,B 0,C 180,E1 -5558.998,E2 -5558.998} C_VEL
LIN {X 0,Y 509.866,Z 286.978,A -85,B 0,C 180,E1 -5561.516,E2 -5561.516} C_VEL
LIN {X 0,Y 509.917,Z 286.962,A -85,B 0,C 180,E1 -5564.819,E2 -5564.819} C_VEL
LIN {X 0,Y 509.906,Z 286.966,A -85,B 0,C 180,E1 -5568.124,E2 -5568.124} C_VEL
LIN {X 0,Y 509.913,Z 286.964,A -85,B 0,C 180,E1 -5571.28,E2 -5571.28} C_VEL
LIN {X 0,Y 509.976,Z 286.956,A -85,B 0,C 180,E1 -5574.464,E2 -5574.464} C_VEL
LIN {X 0,Y 510.059,Z 286.948,A -85,B 0,C 180,E1 -5577.631,E2 -5577.631} C_VEL
LIN {X 0,Y 510.067,Z 286.944,A -85,B 0,C 180,E1 -5580.789,E2 -5580.789} C_VEL
LIN {X 0,Y 509.956,Z 286.957,A -85,B 0,C 180,E1 -5583.16,E2 -5583.16} C_VEL
LIN {X 0,Y 509.957,Z 286.966,A -85,B 0,C 180,E1 -5586.33,E2 -5586.33} C_VEL
LIN {X 0,Y 509.908,Z 286.967,A -85,B 0,C 180,E1 -5588.72,E2 -5588.72} C_VEL
LIN {X 0,Y 509.909,Z 286.964,A -85,B 0,C 180,E1 -5591.931,E2 -5591.931} C_VEL
LIN {X 0,Y 509.899,Z 286.965,A -85,B 0,C 180,E1 -5595.241,E2 -5595.241} C_VEL
LIN {X 0,Y 509.865,Z 286.974,A -85,B 0,C 180,E1 -5598.483,E2 -5598.483} C_VEL
LIN {X 0,Y 509.854,Z 286.976,A -85,B 0,C 180,E1 -5601.001,E2 -5601.001} C_VEL
LIN {X 0,Y 509.868,Z 286.97,A -85,B 0,C 180,E1 -5604.426,E2 -5604.426} C_VEL
LIN {X 0,Y 509.888,Z 286.974,A -85,B 0,C 180,E1 -5607.055,E2 -5607.055} C_VEL
LIN {X 0,Y 509.862,Z 286.969,A -85,B 0,C 180,E1 -5609.751,E2 -5609.751} C_VEL
LIN {X 0,Y 509.877,Z 286.97,A -85,B 0,C 180,E1 -5612.774,E2 -5612.774} C_VEL
LIN {X 0,Y 509.827,Z 286.978,A -85,B 0,C 180,E1 -5615.578,E2 -5615.578} C_VEL
LIN {X 0,Y 509.852,Z 286.969,A -85,B 0,C 180,E1 -5618.338,E2 -5618.338} C_VEL
LIN {X 0,Y 509.859,Z 286.978,A -85,B 0,C 180,E1 -5621.425,E2 -5621.425} C_VEL
LIN {X 0,Y 509.843,Z 286.971,A -85,B 0,C 180,E1 -5624.669,E2 -5624.669} C_VEL
LIN {X 0,Y 509.859,Z 286.972,A -85,B 0,C 180,E1 -5628.103,E2 -5628.103} C_VEL
LIN {X 0,Y 509.849,Z 286.97,A -85,B 0,C 180,E1 -5630.647,E2 -5630.647} C_VEL
LIN {X 0,Y 509.824,Z 286.978,A -85,B 0,C 180,E1 -5633.728,E2 -5633.728} C_VEL
LIN {X 0,Y 509.156,Z 287.06,A -85,B 0,C 180,E1 -5634.388,E2 -5634.388} C_VEL
LIN {X 0,Y 506.344,Z 287.409,A -85,B 0,C 180,E1 -5635.46,E2 -5635.46} C_VEL
LIN {X 0,Y 503.958,Z 287.708,A -85,B 0,C 180,E1 -5636.324,E2 -5636.324} C_VEL
LIN {X 0,Y 502.91,Z 287.835,A -85,B 0,C 180,E1 -5636.99,E2 -5636.99} C_VEL
LIN {X 0,Y 502.812,Z 287.847,A -85,B 0,C 180,E1 -5637.216,E2 -5637.216} C_VEL
LIN {X 0,Y 502.818,Z 287.856,A -85,B 0,C 180,E1 -5640.064,E2 -5640.064} C_VEL
LIN {X 0,Y 502.837,Z 287.847,A -85,B 0,C 180,E1 -5642.532,E2 -5642.532} C_VEL
LIN {X 0,Y 502.807,Z 287.847,A -85,B 0,C 180,E1 -5645.304,E2 -5645.304} C_VEL
LIN {X 0,Y 502.783,Z 287.853,A -85,B 0,C 180,E1 -5647.826,E2 -5647.826} C_VEL
LIN {X 0,Y 502.828,Z 287.854,A -85,B 0,C 180,E1 -5650.399,E2 -5650.399} C_VEL
LIN {X 0,Y 502.831,Z 287.848,A -85,B 0,C 180,E1 -5652.931,E2 -5652.931} C_VEL
LIN {X 0,Y 502.847,Z 287.842,A -85,B 0,C 180,E1 -5655.428,E2 -5655.428} C_VEL
LIN {X 0,Y 502.879,Z 287.848,A -85,B 0,C 180,E1 -5658.716,E2 -5658.716} C_VEL
LIN {X 0,Y 502.882,Z 287.841,A -85,B 0,C 180,E1 -5661.965,E2 -5661.965} C_VEL
LIN {X 0,Y 502.923,Z 287.963,A -85,B 0,C 180,E1 -5665.013,E2 -5665.013} C_VEL
LIN {X 0,Y 503.506,Z 293.942,A -85,B 0,C 180,E1 -5666.197,E2 -5666.197} C_VEL
LIN {X 0,Y 503.256,Z 309.565,A -85,B 0,C 180,E1 -5669.199,E2 -5669.199} C_VEL
LIN {X 0,Y 503.268,Z 310.209,A -85,B 0,C 180,E1 -5669.261,E2 -5669.261} C_VEL
LIN {X 0,Y 505.466,Z 321.844,A -85,B 0,C 180,E1 -5669.501,E2 -5669.501} C_VEL
LIN {X 0,Y 504.827,Z 416.604,A -85,B 0,C 180,E1 -5670.871,E2 -5670.871} C_VEL
LIN {X 0,Y 504.617,Z 429.759,A -85,B 0,C 180,E1 -5671.221,E2 -5671.221} C_VEL
LIN {X 0,Y 504.377,Z 442.899,A -85,B 0,C 180,E1 -5671.745,E2 -5671.745} C_VEL
LIN {X 0,Y 504.09,Z 454.769,A -85,B 0,C 180,E1 -5672.396,E2 -5672.396} C_VEL
LIN {X 0,Y 503.693,Z 466.151,A -85,B 0,C 180,E1 -5673.198,E2 -5673.198} C_VEL
LIN {X 0,Y 503.332,Z 476.418,A -85,B 0,C 180,E1 -5674.102,E2 -5674.102} C_VEL
LIN {X 0,Y 503.027,Z 484.833,A -85,B 0,C 180,E1 -5675.008,E2 -5675.008} C_VEL
LIN {X 0,Y 502.714,Z 493.968,A -85,B 0,C 180,E1 -5676.219,E2 -5676.219} C_VEL
LIN {X 0,Y 502.535,Z 501.321,A -85,B 0,C 180,E1 -5677.431,E2 -5677.431} C_VEL
LIN {X 0,Y 502.323,Z 508.119,A -85,B 0,C 180,E1 -5678.852,E2 -5678.852} C_VEL
LIN {X 0,Y 502.213,Z 512.605,A -85,B 0,C 180,E1 -5680.073,E2 -5680.073} C_VEL
LIN {X 0,Y 502.152,Z 516.598,A -85,B 0,C 180,E1 -5681.564,E2 -5681.564} C_VEL
LIN {X 0,Y 502.021,Z 518.995,A -85,B 0,C 180,E1 -5682.942,E2 -5682.942} C_VEL
LIN {X 0,Y 502.017,Z 519.868,A -85,B 0,C 180,E1 -5683.767,E2 -5683.767} C_VEL
LIN {X 0,Y 502.045,Z 520.367,A -85,B 0,C 180,E1 -5685.003,E2 -5685.003} C_VEL
LIN {X 0,Y 501.981,Z 519.917,A -85,B 0,C 180,E1 -5686.259,E2 -5686.259} C_VEL
LIN {X 0,Y 502.02,Z 519.077,A -85,B 0,C 180,E1 -5687.095,E2 -5687.095} C_VEL
LIN {X 0,Y 502.05,Z 517.786,A -85,B 0,C 180,E1 -5687.935,E2 -5687.935} C_VEL
LIN {X 0,Y 502.151,Z 514.997,A -85,B 0,C 180,E1 -5689.201,E2 -5689.201} C_VEL
LIN {X 0,Y 502.254,Z 511.072,A -85,B 0,C 180,E1 -5690.475,E2 -5690.475} C_VEL
LIN {X 0,Y 502.343,Z 505.868,A -85,B 0,C 180,E1 -5691.76,E2 -5691.76} C_VEL
LIN {X 0,Y 502.582,Z 499.194,A -85,B 0,C 180,E1 -5693.049,E2 -5693.049} C_VEL
LIN {X 0,Y 502.886,Z 490.656,A -85,B 0,C 180,E1 -5694.346,E2 -5694.346} C_VEL
LIN {X 0,Y 503.16,Z 481.787,A -85,B 0,C 180,E1 -5695.435,E2 -5695.435} C_VEL
LIN {X 0,Y 503.543,Z 471.903,A -85,B 0,C 180,E1 -5696.414,E2 -5696.414} C_VEL
LIN {X 0,Y 503.874,Z 460.682,A -85,B 0,C 180,E1 -5697.306,E2 -5697.306} C_VEL
LIN {X 0,Y 504.288,Z 448.649,A -85,B 0,C 180,E1 -5698.056,E2 -5698.056} C_VEL
LIN {X 0,Y 504.541,Z 436.744,A -85,B 0,C 180,E1 -5698.615,E2 -5698.615} C_VEL
LIN {X 0,Y 504.792,Z 423.617,A -85,B 0,C 180,E1 -5699.053,E2 -5699.053} C_VEL
LIN {X 0,Y 504.959,Z 410.526,A -85,B 0,C 180,E1 -5699.322,E2 -5699.322} C_VEL
LIN {X 0,Y 505.458,Z 321.419,A -85,B 0,C 180,E1 -5700.599,E2 -5700.599} C_VEL
LIN {X 0,Y 503.236,Z 309.653,A -85,B 0,C 180,E1 -5700.855,E2 -5700.855} C_VEL
LIN {X 0,Y 503.447,Z 292.922,A -85,B 0,C 180,E1 -5703.943,E2 -5703.943} C_VEL
LIN {X 0,Y 502.778,Z 287.862,A -85,B 0,C 180,E1 -5704.929,E2 -5704.929} C_VEL
LIN {X 0,Y 502.746,Z 287.859,A -85,B 0,C 180,E1 -5708.479,E2 -5708.479} C_VEL
LIN {X 0,Y 502.75,Z 287.861,A -85,B 0,C 180,E1 -5711.071,E2 -5711.071} C_VEL
LIN {X 0,Y 502.765,Z 287.855,A -85,B 0,C 180,E1 -5714.528,E2 -5714.528} C_VEL
LIN {X 0,Y 502.753,Z 287.86,A -85,B 0,C 180,E1 -5717.856,E2 -5717.856} C_VEL
LIN {X 0,Y 502.77,Z 287.856,A -85,B 0,C 180,E1 -5721.021,E2 -5721.021} C_VEL
LIN {X 0,Y 502.751,Z 287.851,A -85,B 0,C 180,E1 -5724.17,E2 -5724.17} C_VEL
LIN {X 0,Y 502.817,Z 287.848,A -85,B 0,C 180,E1 -5726.993,E2 -5726.993} C_VEL
LIN {X 0,Y 502.801,Z 287.854,A -85,B 0,C 180,E1 -5730.064,E2 -5730.064} C_VEL
LIN {X 0,Y 502.798,Z 287.852,A -85,B 0,C 180,E1 -5733.43,E2 -5733.43} C_VEL
LIN {X 0,Y 502.76,Z 287.861,A -85,B 0,C 180,E1 -5736.085,E2 -5736.085} C_VEL
LIN {X 0,Y 502.766,Z 287.851,A -85,B 0,C 180,E1 -5738.688,E2 -5738.688} C_VEL
LIN {X 0,Y 502.811,Z 287.848,A -85,B 0,C 180,E1 -5741.248,E2 -5741.248} C_VEL
LIN {X 0,Y 502.833,Z 287.847,A -85,B 0,C 180,E1 -5744.6,E2 -5744.6} C_VEL
LIN {X 0,Y 502.861,Z 287.846,A -85,B 0,C 180,E1 -5748.039,E2 -5748.039} C_VEL
LIN {X 0,Y 502.858,Z 287.842,A -85,B 0,C 180,E1 -5751.157,E2 -5751.157} C_VEL
LIN {X 0,Y 502.911,Z 287.841,A -85,B 0,C 180,E1 -5754.386,E2 -5754.386} C_VEL
LIN {X 0,Y 503.007,Z 287.821,A -85,B 0,C 180,E1 -5757.598,E2 -5757.598} C_VEL
LIN {X 0,Y 503.008,Z 287.824,A -85,B 0,C 180,E1 -5760,E2 -5760} C_VEL
LIN {X 0,Y 503.008,Z 287.829,A -85,B 0,C 180,E1 -5762.402,E2 -5762.402} C_VEL
LIN {X 0,Y 502.92,Z 287.833,A -85,B 0,C 180,E1 -5765.614,E2 -5765.614} C_VEL
LIN {X 0,Y 502.888,Z 287.836,A -85,B 0,C 180,E1 -5768.034,E2 -5768.034} C_VEL
LIN {X 0,Y 502.867,Z 287.842,A -85,B 0,C 180,E1 -5771.284,E2 -5771.284} C_VEL
LIN {X 0,Y 502.831,Z 287.845,A -85,B 0,C 180,E1 -5774.571,E2 -5774.571} C_VEL
LIN {X 0,Y 502.848,Z 287.841,A -85,B 0,C 180,E1 -5777.908,E2 -5777.908} C_VEL
LIN {X 0,Y 502.815,Z 287.849,A -85,B 0,C 180,E1 -5780.537,E2 -5780.537} C_VEL
LIN {X 0,Y 502.784,Z 287.856,A -85,B 0,C 180,E1 -5783.041,E2 -5783.041} C_VEL
LIN {X 0,Y 502.83,Z 287.847,A -85,B 0,C 180,E1 -5785.676,E2 -5785.676} C_VEL
LIN {X 0,Y 502.83,Z 287.842,A -85,B 0,C 180,E1 -5788.374,E2 -5788.374} C_VEL
LIN {X 0,Y 502.786,Z 287.854,A -85,B 0,C 180,E1 -5791.501,E2 -5791.501} C_VEL
LIN {X 0,Y 502.797,Z 287.851,A -85,B 0,C 180,E1 -5794.446,E2 -5794.446} C_VEL
LIN {X 0,Y 502.774,Z 287.858,A -85,B 0,C 180,E1 -5797.18,E2 -5797.18} C_VEL
LIN {X 0,Y 502.803,Z 287.852,A -85,B 0,C 180,E1 -5800.014,E2 -5800.014} C_VEL
LIN {X 0,Y 502.794,Z 287.85,A -85,B 0,C 180,E1 -5802.201,E2 -5802.201} C_VEL
LIN {X 0,Y 502.793,Z 287.853,A -85,B 0,C 180,E1 -5805.47,E2 -5805.47} C_VEL
LIN {X 0,Y 502.828,Z 287.852,A -85,B 0,C 180,E1 -5807.866,E2 -5807.866} C_VEL
LIN {X 0,Y 502.804,Z 287.849,A -85,B 0,C 180,E1 -5811.026,E2 -5811.026} C_VEL
LIN {X 0,Y 502.778,Z 287.858,A -85,B 0,C 180,E1 -5814.169,E2 -5814.169} C_VEL
LIN {X 0,Y 502.827,Z 287.846,A -85,B 0,C 180,E1 -5816.995,E2 -5816.995} C_VEL
LIN {X 0,Y 502.811,Z 287.855,A -85,B 0,C 180,E1 -5820.066,E2 -5820.066} C_VEL
LIN {X 0,Y 502.831,Z 287.851,A -85,B 0,C 180,E1 -5822.535,E2 -5822.535} C_VEL
LIN {X 0,Y 502.865,Z 287.911,A -85,B 0,C 180,E1 -5824.954,E2 -5824.954} C_VEL
LIN {X 0,Y 504.49,Z 297.154,A -85,B 0,C 180,E1 -5826.563,E2 -5826.563} C_VEL
LIN {X 0,Y 504.141,Z 312.01,A -85,B 0,C 180,E1 -5828.979,E2 -5828.979} C_VEL
LIN {X 0,Y 503.582,Z 331.683,A -85,B 0,C 180,E1 -5832.121,E2 -5832.121} C_VEL
LIN {X 0,Y 503.262,Z 345.008,A -85,B 0,C 180,E1 -5834.195,E2 -5834.195} C_VEL
LIN {X 0,Y 505.369,Z 358.914,A -85,B 0,C 180,E1 -5834.464,E2 -5834.464} C_VEL
LIN {X 0,Y 504.812,Z 452.953,A -85,B 0,C 180,E1 -5835.823,E2 -5835.823} C_VEL
LIN {X 0,Y 504.544,Z 466.323,A -85,B 0,C 180,E1 -5836.175,E2 -5836.175} C_VEL
LIN {X 0,Y 504.206,Z 479.673,A -85,B 0,C 180,E1 -5836.705,E2 -5836.705} C_VEL
LIN {X 0,Y 503.897,Z 491.98,A -85,B 0,C 180,E1 -5837.383,E2 -5837.383} C_VEL
LIN {X 0,Y 503.547,Z 502.514,A -85,B 0,C 180,E1 -5838.121,E2 -5838.121} C_VEL
LIN {X 0,Y 503.21,Z 512.993,A -85,B 0,C 180,E1 -5839.032,E2 -5839.032} C_VEL
LIN {X 0,Y 502.871,Z 521.559,A -85,B 0,C 180,E1 -5839.94,E2 -5839.94} C_VEL
LIN {X 0,Y 502.619,Z 529.467,A -85,B 0,C 180,E1 -5840.951,E2 -5840.951} C_VEL
LIN {X 0,Y 502.398,Z 537.192,A -85,B 0,C 180,E1 -5842.162,E2 -5842.162} C_VEL
LIN {X 0,Y 502.235,Z 543.902,A -85,B 0,C 180,E1 -5843.483,E2 -5843.483} C_VEL
LIN {X 0,Y 502.174,Z 549.052,A -85,B 0,C 180,E1 -5844.782,E2 -5844.782} C_VEL
LIN {X 0,Y 502.139,Z 552.674,A -85,B 0,C 180,E1 -5845.988,E2 -5845.988} C_VEL
LIN {X 0,Y 502.12,Z 554.542,A -85,B 0,C 180,E1 -5846.792,E2 -5846.792} C_VEL
LIN {X 0,Y 502.091,Z 555.943,A -85,B 0,C 180,E1 -5847.595,E2 -5847.595} C_VEL
LIN {X 0,Y 501.99,Z 557.551,A -85,B 0,C 180,E1 -5849.199,E2 -5849.199} C_VEL
LIN {X 0,Y 501.983,Z 557.769,A -85,B 0,C 180,E1 -5850.001,E2 -5850.001} C_VEL
LIN {X 0,Y 502.036,Z 556.948,A -85,B 0,C 180,E1 -5851.606,E2 -5851.606} C_VEL
LIN {X 0,Y 502.091,Z 555.954,A -85,B 0,C 180,E1 -5852.408,E2 -5852.408} C_VEL
LIN {X 0,Y 502.121,Z 554.556,A -85,B 0,C 180,E1 -5853.211,E2 -5853.211} C_VEL
LIN {X 0,Y 502.102,Z 551.613,A -85,B 0,C 180,E1 -5854.416,E2 -5854.416} C_VEL
LIN {X 0,Y 502.21,Z 547.632,A -85,B 0,C 180,E1 -5855.623,E2 -5855.623} C_VEL
LIN {X 0,Y 502.332,Z 541.608,A -85,B 0,C 180,E1 -5857.013,E2 -5857.013} C_VEL
LIN {X 0,Y 502.478,Z 534.812,A -85,B 0,C 180,E1 -5858.244,E2 -5858.244} C_VEL
LIN {X 0,Y 502.717,Z 526.508,A -85,B 0,C 180,E1 -5859.456,E2 -5859.456} C_VEL
LIN {X 0,Y 502.975,Z 517.994,A -85,B 0,C 180,E1 -5860.467,E2 -5860.467} C_VEL
LIN {X 0,Y 503.414,Z 507.479,A -85,B 0,C 180,E1 -5861.476,E2 -5861.476} C_VEL
LIN {X 0,Y 503.685,Z 497.156,A -85,B 0,C 180,E1 -5862.281,E2 -5862.281} C_VEL
LIN {X 0,Y 504.056,Z 485.664,A -85,B 0,C 180,E1 -5862.994,E2 -5862.994} C_VEL
LIN {X 0,Y 504.339,Z 473.931,A -85,B 0,C 180,E1 -5863.55,E2 -5863.55} C_VEL
LIN {X 0,Y 504.687,Z 460.416,A -85,B 0,C 180,E1 -5864.003,E2 -5864.003} C_VEL
LIN {X 0,Y 504.907,Z 446.922,A -85,B 0,C 180,E1 -5864.279,E2 -5864.279} C_VEL
LIN {X 0,Y 505.321,Z 358.723,A -85,B 0,C 180,E1 -5865.542,E2 -5865.542} C_VEL
LIN {X 0,Y 503.249,Z 344.819,A -85,B 0,C 180,E1 -5865.823,E2 -5865.823} C_VEL
LIN {X 0,Y 503.771,Z 325.304,A -85,B 0,C 180,E1 -5868.928,E2 -5868.928} C_VEL
LIN {X 0,Y 504.384,Z 305.622,A -85,B 0,C 180,E1 -5872.1,E2 -5872.1} C_VEL
LIN {X 0,Y 504.563,Z 297.366,A -85,B 0,C 180,E1 -5873.447,E2 -5873.447} C_VEL
LIN {X 0,Y 502.876,Z 287.846,A -85,B 0,C 180,E1 -5875.109,E2 -5875.109} C_VEL
LIN {X 0,Y 502.833,Z 287.849,A -85,B 0,C 180,E1 -5877.468,E2 -5877.468} C_VEL
LIN {X 0,Y 502.815,Z 287.856,A -85,B 0,C 180,E1 -5880.212,E2 -5880.212} C_VEL
LIN {X 0,Y 502.835,Z 287.844,A -85,B 0,C 180,E1 -5883.032,E2 -5883.032} C_VEL
LIN {X 0,Y 502.779,Z 287.855,A -85,B 0,C 180,E1 -5885.952,E2 -5885.952} C_VEL
LIN {X 0,Y 502.8,Z 287.85,A -85,B 0,C 180,E1 -5888.977,E2 -5888.977} C_VEL
LIN {X 0,Y 502.825,Z 287.847,A -85,B 0,C 180,E1 -5891.066,E2 -5891.066} C_VEL
LIN {X 0,Y 502.792,Z 287.858,A -85,B 0,C 180,E1 -5894.53,E2 -5894.53} C_VEL
LIN {X 0,Y 502.801,Z 287.848,A -85,B 0,C 180,E1 -5897.861,E2 -5897.861} C_VEL
LIN {X 0,Y 502.806,Z 287.854,A -85,B 0,C 180,E1 -5901.024,E2 -5901.024} C_VEL
LIN {X 0,Y 502.78,Z 287.851,A -85,B 0,C 180,E1 -5904.169,E2 -5904.169} C_VEL
LIN {X 0,Y 502.808,Z 287.857,A -85,B 0,C 180,E1 -5906.999,E2 -5906.999} C_VEL
LIN {X 0,Y 502.821,Z 287.845,A -85,B 0,C 180,E1 -5910.065,E2 -5910.065} C_VEL
LIN {X 0,Y 502.836,Z 287.845,A -85,B 0,C 180,E1 -5912.533,E2 -5912.533} C_VEL
LIN {X 0,Y 502.831,Z 287.854,A -85,B 0,C 180,E1 -5915.3,E2 -5915.3} C_VEL
LIN {X 0,Y 502.785,Z 287.853,A -85,B 0,C 180,E1 -5917.826,E2 -5917.826} C_VEL
LIN {X 0,Y 502.828,Z 287.845,A -85,B 0,C 180,E1 -5920.4,E2 -5920.4} C_VEL
LIN {X 0,Y 502.823,Z 287.847,A -85,B 0,C 180,E1 -5922.931,E2 -5922.931} C_VEL
LIN {X 0,Y 502.849,Z 287.849,A -85,B 0,C 180,E1 -5925.429,E2 -5925.429} C_VEL
LIN {X 0,Y 502.882,Z 287.838,A -85,B 0,C 180,E1 -5928.717,E2 -5928.717} C_VEL
LIN {X 0,Y 502.905,Z 287.843,A -85,B 0,C 180,E1 -5931.967,E2 -5931.967} C_VEL
LIN {X 0,Y 502.93,Z 287.835,A -85,B 0,C 180,E1 -5934.386,E2 -5934.386} C_VEL
LIN {X 0,Y 503.029,Z 287.823,A -85,B 0,C 180,E1 -5937.598,E2 -5937.598} C_VEL
LIN {X 0,Y 503.016,Z 287.822,A -85,B 0,C 180,E1 -5940.8,E2 -5940.8} C_VEL
LIN {X 0,Y 502.899,Z 287.836,A -85,B 0,C 180,E1 -5943.204,E2 -5943.204} C_VEL
LIN {X 0,Y 502.909,Z 287.843,A -85,B 0,C 180,E1 -5946.419,E2 -5946.419} C_VEL
LIN {X 0,Y 502.868,Z 287.843,A -85,B 0,C 180,E1 -5948.843,E2 -5948.843} C_VEL
LIN {X 0,Y 502.85,Z 287.845,A -85,B 0,C 180,E1 -5952.101,E2 -5952.101} C_VEL
LIN {X 0,Y 502.854,Z 287.842,A -85,B 0,C 180,E1 -5955.399,E2 -5955.399} C_VEL
LIN {X 0,Y 502.83,Z 287.854,A -85,B 0,C 180,E1 -5958.752,E2 -5958.752} C_VEL
LIN {X 0,Y 502.787,Z 287.852,A -85,B 0,C 180,E1 -5961.311,E2 -5961.311} C_VEL
LIN {X 0,Y 502.789,Z 287.849,A -85,B 0,C 180,E1 -5963.914,E2 -5963.914} C_VEL
LIN {X 0,Y 502.869,Z 287.843,A -85,B 0,C 180,E1 -5966.566,E2 -5966.566} C_VEL
LIN {X 0,Y 502.828,Z 287.851,A -85,B 0,C 180,E1 -5969.287,E2 -5969.287} C_VEL
LIN {X 0,Y 502.787,Z 287.85,A -85,B 0,C 180,E1 -5972.084,E2 -5972.084} C_VEL
LIN {X 0,Y 502.801,Z 287.853,A -85,B 0,C 180,E1 -5974.965,E2 -5974.965} C_VEL
LIN {X 0,Y 502.797,Z 287.849,A -85,B 0,C 180,E1 -5978.485,E2 -5978.485} C_VEL
LIN {X 0,Y 502.824,Z 287.849,A -85,B 0,C 180,E1 -5981.065,E2 -5981.065} C_VEL
LIN {X 0,Y 502.789,Z 287.849,A -85,B 0,C 180,E1 -5984.529,E2 -5984.529} C_VEL
LIN {X 0,Y 502.799,Z 287.855,A -85,B 0,C 180,E1 -5987.86,E2 -5987.86} C_VEL
LIN {X 0,Y 502.804,Z 287.848,A -85,B 0,C 180,E1 -5991.023,E2 -5991.023} C_VEL
LIN {X 0,Y 502.778,Z 287.856,A -85,B 0,C 180,E1 -5994.168,E2 -5994.168} C_VEL
LIN {X 0,Y 502.812,Z 287.847,A -85,B 0,C 180,E1 -5997.216,E2 -5997.216} C_VEL
LIN {X 0,Y 502.11,Z 287.942,A -85,B 0,C 180,E1 -5997.884,E2 -5997.884} C_VEL
LIN {X 0,Y 499.245,Z 288.298,A -85,B 0,C 180,E1 -5998.97,E2 -5998.97} C_VEL
LIN {X 0,Y 496.851,Z 288.595,A -85,B 0,C 180,E1 -5999.845,E2 -5999.845} C_VEL
LIN {X 0,Y 495.835,Z 288.72,A -85,B 0,C 180,E1 -6000.521,E2 -6000.521} C_VEL
LIN {X 0,Y 495.757,Z 288.727,A -85,B 0,C 180,E1 -6000.749,E2 -6000.749} C_VEL
LIN {X 0,Y 495.827,Z 288.717,A -85,B 0,C 180,E1 -6003.25,E2 -6003.25} C_VEL
LIN {X 0,Y 495.746,Z 288.731,A -85,B 0,C 180,E1 -6006.612,E2 -6006.612} C_VEL
LIN {X 0,Y 495.782,Z 288.722,A -85,B 0,C 180,E1 -6009.323,E2 -6009.323} C_VEL
LIN {X 0,Y 495.796,Z 288.722,A -85,B 0,C 180,E1 -6011.828,E2 -6011.828} C_VEL
LIN {X 0,Y 495.827,Z 288.727,A -85,B 0,C 180,E1 -6014.547,E2 -6014.547} C_VEL
LIN {X 0,Y 495.831,Z 288.717,A -85,B 0,C 180,E1 -6017.964,E2 -6017.964} C_VEL
LIN {X 0,Y 495.836,Z 288.723,A -85,B 0,C 180,E1 -6021.029,E2 -6021.029} C_VEL
LIN {X 0,Y 495.862,Z 288.719,A -85,B 0,C 180,E1 -6023.488,E2 -6023.488} C_VEL
LIN {X 0,Y 495.902,Z 288.765,A -85,B 0,C 180,E1 -6024.866,E2 -6024.866} C_VEL
LIN {X 0,Y 496.519,Z 295.141,A -85,B 0,C 180,E1 -6026.144,E2 -6026.144} C_VEL
LIN {X 0,Y 496.272,Z 309.958,A -85,B 0,C 180,E1 -6029.01,E2 -6029.01} C_VEL
LIN {X 0,Y 498.613,Z 322.546,A -85,B 0,C 180,E1 -6029.292,E2 -6029.292} C_VEL
LIN {X 0,Y 497.966,Z 417.094,A -85,B 0,C 180,E1 -6030.681,E2 -6030.681} C_VEL
LIN {X 0,Y 497.744,Z 430.177,A -85,B 0,C 180,E1 -6031.035,E2 -6031.035} C_VEL
LIN {X 0,Y 497.487,Z 443.286,A -85,B 0,C 180,E1 -6031.567,E2 -6031.567} C_VEL
LIN {X 0,Y 497.163,Z 455.135,A -85,B 0,C 180,E1 -6032.227,E2 -6032.227} C_VEL
LIN {X 0,Y 496.741,Z 466.508,A -85,B 0,C 180,E1 -6033.04,E2 -6033.04} C_VEL
LIN {X 0,Y 496.359,Z 476.765,A -85,B 0,C 180,E1 -6033.957,E2 -6033.957} C_VEL
LIN {X 0,Y 496.019,Z 485.175,A -85,B 0,C 180,E1 -6034.875,E2 -6034.875} C_VEL
LIN {X 0,Y 495.682,Z 494.292,A -85,B 0,C 180,E1 -6036.103,E2 -6036.103} C_VEL
LIN {X 0,Y 495.503,Z 501.631,A -85,B 0,C 180,E1 -6037.333,E2 -6037.333} C_VEL
LIN {X 0,Y 495.298,Z 507.55,A -85,B 0,C 180,E1 -6038.567,E2 -6038.567} C_VEL
LIN {X 0,Y 495.125,Z 512.235,A -85,B 0,C 180,E1 -6039.806,E2 -6039.806} C_VEL
LIN {X 0,Y 495.098,Z 515.8,A -85,B 0,C 180,E1 -6041.047,E2 -6041.047} C_VEL
LIN {X 0,Y 494.953,Z 518.36,A -85,B 0,C 180,E1 -6042.296,E2 -6042.296} C_VEL
LIN {X 0,Y 494.938,Z 519.537,A -85,B 0,C 180,E1 -6043.131,E2 -6043.131} C_VEL
LIN {X 0,Y 494.927,Z 520.264,A -85,B 0,C 180,E1 -6043.968,E2 -6043.968} C_VEL
LIN {X 0,Y 494.958,Z 520.631,A -85,B 0,C 180,E1 -6045.084,E2 -6045.084} C_VEL
LIN {X 0,Y 494.889,Z 519.997,A -85,B 0,C 180,E1 -6046.499,E2 -6046.499} C_VEL
LIN {X 0,Y 494.959,Z 518.104,A -85,B 0,C 180,E1 -6047.947,E2 -6047.947} C_VEL
LIN {X 0,Y 495.099,Z 514.68,A -85,B 0,C 180,E1 -6049.485,E2 -6049.485} C_VEL
LIN {X 0,Y 495.199,Z 510.548,A -85,B 0,C 180,E1 -6050.78,E2 -6050.78} C_VEL
LIN {X 0,Y 495.337,Z 505.083,A -85,B 0,C 180,E1 -6052.084,E2 -6052.084} C_VEL
LIN {X 0,Y 495.589,Z 498.083,A -85,B 0,C 180,E1 -6053.394,E2 -6053.394} C_VEL
LIN {X 0,Y 495.898,Z 489.759,A -85,B 0,C 180,E1 -6054.641,E2 -6054.641} C_VEL
LIN {X 0,Y 496.246,Z 480.969,A -85,B 0,C 180,E1 -6055.702,E2 -6055.702} C_VEL
LIN {X 0,Y 496.624,Z 470.796,A -85,B 0,C 180,E1 -6056.698,E2 -6056.698} C_VEL
LIN {X 0,Y 496.979,Z 459.799,A -85,B 0,C 180,E1 -6057.565,E2 -6057.565} C_VEL
LIN {X 0,Y 497.409,Z 447.698,A -85,B 0,C 180,E1 -6058.306,E2 -6058.306} C_VEL
LIN {X 0,Y 497.684,Z 436.31,A -85,B 0,C 180,E1 -6058.837,E2 -6058.837} C_VEL
LIN {X 0,Y 497.957,Z 423.523,A -85,B 0,C 180,E1 -6059.263,E2 -6059.263} C_VEL
LIN {X 0,Y 498.097,Z 409.876,A -85,B 0,C 180,E1 -6059.54,E2 -6059.54} C_VEL
LIN {X 0,Y 498.611,Z 322.061,A -85,B 0,C 180,E1 -6060.816,E2 -6060.816} C_VEL
LIN {X 0,Y 496.27,Z 309.813,A -85,B 0,C 180,E1 -6061.099,E2 -6061.099} C_VEL
LIN {X 0,Y 496.493,Z 294.296,A -85,B 0,C 180,E1 -6063.994,E2 -6063.994} C_VEL
LIN {X 0,Y 495.732,Z 288.739,A -85,B 0,C 180,E1 -6065.099,E2 -6065.099} C_VEL
LIN {X 0,Y 495.723,Z 288.737,A -85,B 0,C 180,E1 -6068.763,E2 -6068.763} C_VEL
LIN {X 0,Y 495.711,Z 288.737,A -85,B 0,C 180,E1 -6071.783,E2 -6071.783} C_VEL
LIN {X 0,Y 495.723,Z 288.737,A -85,B 0,C 180,E1 -6075.14,E2 -6075.14} C_VEL
LIN {X 0,Y 495.713,Z 288.734,A -85,B 0,C 180,E1 -6078.215,E2 -6078.215} C_VEL
LIN {X 0,Y 495.727,Z 288.736,A -85,B 0,C 180,E1 -6081.234,E2 -6081.234} C_VEL
LIN {X 0,Y 495.725,Z 288.724,A -85,B 0,C 180,E1 -6084.461,E2 -6084.461} C_VEL
LIN {X 0,Y 495.752,Z 288.733,A -85,B 0,C 180,E1 -6087.405,E2 -6087.405} C_VEL
LIN {X 0,Y 495.749,Z 288.73,A -85,B 0,C 180,E1 -6090.253,E2 -6090.253} C_VEL
LIN {X 0,Y 495.745,Z 288.729,A -85,B 0,C 180,E1 -6093.265,E2 -6093.265} C_VEL
LIN {X 0,Y 495.727,Z 288.731,A -85,B 0,C 180,E1 -6096.612,E2 -6096.612} C_VEL
LIN {X 0,Y 495.764,Z 288.723,A -85,B 0,C 180,E1 -6099.324,E2 -6099.324} C_VEL
LIN {X 0,Y 495.766,Z 288.731,A -85,B 0,C 180,E1 -6101.828,E2 -6101.828} C_VEL
LIN {X 0,Y 495.808,Z 288.723,A -85,B 0,C 180,E1 -6104.548,E2 -6104.548} C_VEL
LIN {X 0,Y 495.813,Z 288.723,A -85,B 0,C 180,E1 -6107.965,E2 -6107.965} C_VEL
LIN {X 0,Y 495.826,Z 288.718,A -85,B 0,C 180,E1 -6111.03,E2 -6111.03} C_VEL
LIN {X 0,Y 495.866,Z 288.717,A -85,B 0,C 180,E1 -6114.306,E2 -6114.306} C_VEL
LIN {X 0,Y 495.976,Z 288.696,A -85,B 0,C 180,E1 -6117.564,E2 -6117.564} C_VEL
LIN {X 0,Y 495.979,Z 288.699,A -85,B 0,C 180,E1 -6120,E2 -6120} C_VEL
LIN {X 0,Y 495.977,Z 288.704,A -85,B 0,C 180,E1 -6122.437,E2 -6122.437} C_VEL
LIN {X 0,Y 495.876,Z 288.711,A -85,B 0,C 180,E1 -6125.694,E2 -6125.694} C_VEL
LIN {X 0,Y 495.859,Z 288.713,A -85,B 0,C 180,E1 -6128.148,E2 -6128.148} C_VEL
LIN {X 0,Y 495.841,Z 288.716,A -85,B 0,C 180,E1 -6131.446,E2 -6131.446} C_VEL
LIN {X 0,Y 495.776,Z 288.727,A -85,B 0,C 180,E1 -6134.783,E2 -6134.783} C_VEL
LIN {X 0,Y 495.772,Z 288.726,A -85,B 0,C 180,E1 -6137.319,E2 -6137.319} C_VEL
LIN {X 0,Y 495.758,Z 288.725,A -85,B 0,C 180,E1 -6139.891,E2 -6139.891} C_VEL
LIN {X 0,Y 495.745,Z 288.734,A -85,B 0,C 180,E1 -6142.861,E2 -6142.861} C_VEL
LIN {X 0,Y 495.787,Z 288.723,A -85,B 0,C 180,E1 -6146.068,E2 -6146.068} C_VEL
LIN {X 0,Y 495.767,Z 288.725,A -85,B 0,C 180,E1 -6148.815,E2 -6148.815} C_VEL
LIN {X 0,Y 495.748,Z 288.728,A -85,B 0,C 180,E1 -6151.727,E2 -6151.727} C_VEL
LIN {X 0,Y 495.766,Z 288.728,A -85,B 0,C 180,E1 -6154.697,E2 -6154.697} C_VEL
LIN {X 0,Y 495.726,Z 288.738,A -85,B 0,C 180,E1 -6157.562,E2 -6157.562} C_VEL
LIN {X 0,Y 495.772,Z 288.727,A -85,B 0,C 180,E1 -6160.051,E2 -6160.051} C_VEL
LIN {X 0,Y 495.725,Z 288.731,A -85,B 0,C 180,E1 -6162.884,E2 -6162.884} C_VEL
LIN {X 0,Y 495.729,Z 288.731,A -85,B 0,C 180,E1 -6166.001,E2 -6166.001} C_VEL
LIN {X 0,Y 495.762,Z 288.727,A -85,B 0,C 180,E1 -6168.707,E2 -6168.707} C_VEL
LIN {X 0,Y 495.749,Z 288.731,A -85,B 0,C 180,E1 -6171.41,E2 -6171.41} C_VEL
LIN {X 0,Y 495.75,Z 288.731,A -85,B 0,C 180,E1 -6174.464,E2 -6174.464} C_VEL
LIN {X 0,Y 495.763,Z 288.729,A -85,B 0,C 180,E1 -6177.407,E2 -6177.407} C_VEL
LIN {X 0,Y 495.762,Z 288.731,A -85,B 0,C 180,E1 -6180.255,E2 -6180.255} C_VEL
LIN {X 0,Y 495.821,Z 288.723,A -85,B 0,C 180,E1 -6183.252,E2 -6183.252} C_VEL
LIN {X 0,Y 495.822,Z 288.783,A -85,B 0,C 180,E1 -6184.752,E2 -6184.752} C_VEL
LIN {X 0,Y 497.589,Z 298.672,A -85,B 0,C 180,E1 -6186.508,E2 -6186.508} C_VEL
LIN {X 0,Y 497.149,Z 314.011,A -85,B 0,C 180,E1 -6189.034,E2 -6189.034} C_VEL
LIN {X 0,Y 496.564,Z 332.743,A -85,B 0,C 180,E1 -6192.073,E2 -6192.073} C_VEL
LIN {X 0,Y 496.239,Z 344.487,A -85,B 0,C 180,E1 -6193.956,E2 -6193.956} C_VEL
LIN {X 0,Y 498.494,Z 360.623,A -85,B 0,C 180,E1 -6194.27,E2 -6194.27} C_VEL
LIN {X 0,Y 497.949,Z 452.758,A -85,B 0,C 180,E1 -6195.624,E2 -6195.624} C_VEL
LIN {X 0,Y 497.636,Z 466.087,A -85,B 0,C 180,E1 -6195.979,E2 -6195.979} C_VEL
LIN {X 0,Y 497.288,Z 479.414,A -85,B 0,C 180,E1 -6196.517,E2 -6196.517} C_VEL
LIN {X 0,Y 496.978,Z 490.585,A -85,B 0,C 180,E1 -6197.131,E2 -6197.131} C_VEL
LIN {X 0,Y 496.549,Z 502.231,A -85,B 0,C 180,E1 -6197.951,E2 -6197.951} C_VEL
LIN {X 0,Y 496.201,Z 512.71,A -85,B 0,C 180,E1 -6198.875,E2 -6198.875} C_VEL
LIN {X 0,Y 495.846,Z 521.279,A -85,B 0,C 180,E1 -6199.796,E2 -6199.796} C_VEL
LIN {X 0,Y 495.562,Z 529.189,A -85,B 0,C 180,E1 -6200.821,E2 -6200.821} C_VEL
LIN {X 0,Y 495.34,Z 536.917,A -85,B 0,C 180,E1 -6202.05,E2 -6202.05} C_VEL
LIN {X 0,Y 495.163,Z 544.041,A -85,B 0,C 180,E1 -6203.482,E2 -6203.482} C_VEL
LIN {X 0,Y 495.105,Z 548.783,A -85,B 0,C 180,E1 -6204.707,E2 -6204.707} C_VEL
LIN {X 0,Y 495.032,Z 552.405,A -85,B 0,C 180,E1 -6205.931,E2 -6205.931} C_VEL
LIN {X 0,Y 495.041,Z 554.275,A -85,B 0,C 180,E1 -6206.746,E2 -6206.746} C_VEL
LIN {X 0,Y 494.997,Z 555.676,A -85,B 0,C 180,E1 -6207.56,E2 -6207.56} C_VEL
LIN {X 0,Y 494.962,Z 556.676,A -85,B 0,C 180,E1 -6208.374,E2 -6208.374} C_VEL
LIN {X 0,Y 494.901,Z 557.505,A -85,B 0,C 180,E1 -6210.001,E2 -6210.001} C_VEL
LIN {X 0,Y 494.962,Z 556.685,A -85,B 0,C 180,E1 -6211.629,E2 -6211.629} C_VEL
LIN {X 0,Y 494.998,Z 555.69,A -85,B 0,C 180,E1 -6212.442,E2 -6212.442} C_VEL
LIN {X 0,Y 495.042,Z 554.293,A -85,B 0,C 180,E1 -6213.257,E2 -6213.257} C_VEL
LIN {X 0,Y 495.008,Z 551.349,A -85,B 0,C 180,E1 -6214.48,E2 -6214.48} C_VEL
LIN {X 0,Y 495.126,Z 547.368,A -85,B 0,C 180,E1 -6215.703,E2 -6215.703} C_VEL
LIN {X 0,Y 495.257,Z 541.24,A -85,B 0,C 180,E1 -6217.134,E2 -6217.134} C_VEL
LIN {X 0,Y 495.426,Z 534.545,A -85,B 0,C 180,E1 -6218.362,E2 -6218.362} C_VEL
LIN {X 0,Y 495.68,Z 526.24,A -85,B 0,C 180,E1 -6219.591,E2 -6219.591} C_VEL
LIN {X 0,Y 495.971,Z 517.724,A -85,B 0,C 180,E1 -6220.616,E2 -6220.616} C_VEL
LIN {X 0,Y 496.437,Z 507.207,A -85,B 0,C 180,E1 -6221.64,E2 -6221.64} C_VEL
LIN {X 0,Y 496.756,Z 495.915,A -85,B 0,C 180,E1 -6222.525,E2 -6222.525} C_VEL
LIN {X 0,Y 497.107,Z 485.385,A -85,B 0,C 180,E1 -6223.179,E2 -6223.179} C_VEL
LIN {X 0,Y 497.425,Z 473.632,A -85,B 0,C 180,E1 -6223.742,E2 -6223.742} C_VEL
LIN {X 0,Y 497.811,Z 460.09,A -85,B 0,C 180,E1 -6224.2,E2 -6224.2} C_VEL
LIN {X 0,Y 498.04,Z 446.516,A -85,B 0,C 180,E1 -6224.481,E2 -6224.481} C_VEL
LIN {X 0,Y 498.439,Z 358.923,A -85,B 0,C 180,E1 -6225.753,E2 -6225.753} C_VEL
LIN {X 0,Y 496.256,Z 344.635,A -85,B 0,C 180,E1 -6226.037,E2 -6226.037} C_VEL
LIN {X 0,Y 496.833,Z 325.028,A -85,B 0,C 180,E1 -6229.202,E2 -6229.202} C_VEL
LIN {X 0,Y 497.478,Z 305.299,A -85,B 0,C 180,E1 -6232.424,E2 -6232.424} C_VEL
LIN {X 0,Y 497.633,Z 298.839,A -85,B 0,C 180,E1 -6233.493,E2 -6233.493} C_VEL
LIN {X 0,Y 495.827,Z 288.725,A -85,B 0,C 180,E1 -6235.278,E2 -6235.278} C_VEL
LIN {X 0,Y 495.782,Z 288.732,A -85,B 0,C 180,E1 -6237.892,E2 -6237.892} C_VEL
LIN {X 0,Y 495.758,Z 288.728,A -85,B 0,C 180,E1 -6240.688,E2 -6240.688} C_VEL
LIN {X 0,Y 495.757,Z 288.726,A -85,B 0,C 180,E1 -6243.565,E2 -6243.565} C_VEL
LIN {X 0,Y 495.734,Z 288.735,A -85,B 0,C 180,E1 -6246.544,E2 -6246.544} C_VEL
LIN {X 0,Y 495.755,Z 288.726,A -85,B 0,C 180,E1 -6249.639,E2 -6249.639} C_VEL
LIN {X 0,Y 495.743,Z 288.736,A -85,B 0,C 180,E1 -6252.507,E2 -6252.507} C_VEL
LIN {X 0,Y 495.743,Z 288.73,A -85,B 0,C 180,E1 -6255.141,E2 -6255.141} C_VEL
LIN {X 0,Y 495.762,Z 288.727,A -85,B 0,C 180,E1 -6258.219,E2 -6258.219} C_VEL
LIN {X 0,Y 495.755,Z 288.727,A -85,B 0,C 180,E1 -6261.409,E2 -6261.409} C_VEL
LIN {X 0,Y 495.752,Z 288.729,A -85,B 0,C 180,E1 -6264.462,E2 -6264.462} C_VEL
LIN {X 0,Y 495.757,Z 288.729,A -85,B 0,C 180,E1 -6267.405,E2 -6267.405} C_VEL
LIN {X 0,Y 495.772,Z 288.724,A -85,B 0,C 180,E1 -6270.254,E2 -6270.254} C_VEL
LIN {X 0,Y 495.829,Z 288.726,A -85,B 0,C 180,E1 -6273.251,E2 -6273.251} C_VEL
LIN {X 0,Y 495.752,Z 288.729,A -85,B 0,C 180,E1 -6275.725,E2 -6275.725} C_VEL
LIN {X 0,Y 495.748,Z 288.727,A -85,B 0,C 180,E1 -6278.371,E2 -6278.371} C_VEL
LIN {X 0,Y 495.787,Z 288.724,A -85,B 0,C 180,E1 -6280.971,E2 -6280.971} C_VEL
LIN {X 0,Y 495.813,Z 288.719,A -85,B 0,C 180,E1 -6284.376,E2 -6284.376} C_VEL
LIN {X 0,Y 495.784,Z 288.722,A -85,B 0,C 180,E1 -6286.891,E2 -6286.891} C_VEL
LIN {X 0,Y 495.777,Z 288.727,A -85,B 0,C 180,E1 -6289.38,E2 -6289.38} C_VEL
LIN {X 0,Y 495.876,Z 288.72,A -85,B 0,C 180,E1 -6291.852,E2 -6291.852} C_VEL
LIN {X 0,Y 495.84,Z 288.715,A -85,B 0,C 180,E1 -6295.121,E2 -6295.121} C_VEL
LIN {X 0,Y 495.997,Z 288.698,A -85,B 0,C 180,E1 -6297.564,E2 -6297.564} C_VEL
LIN {X 0,Y 495.968,Z 288.7,A -85,B 0,C 180,E1 -6300.812,E2 -6300.812} C_VEL
LIN {X 0,Y 495.996,Z 288.701,A -85,B 0,C 180,E1 -6302.436,E2 -6302.436} C_VEL
LIN {X 0,Y 495.891,Z 288.71,A -85,B 0,C 180,E1 -6305.693,E2 -6305.693} C_VEL
LIN {X 0,Y 495.841,Z 288.721,A -85,B 0,C 180,E1 -6308.148,E2 -6308.148} C_VEL
LIN {X 0,Y 495.856,Z 288.713,A -85,B 0,C 180,E1 -6311.445,E2 -6311.445} C_VEL
LIN {X 0,Y 495.798,Z 288.727,A -85,B 0,C 180,E1 -6314.782,E2 -6314.782} C_VEL
LIN {X 0,Y 495.768,Z 288.725,A -85,B 0,C 180,E1 -6317.319,E2 -6317.319} C_VEL
LIN {X 0,Y 495.775,Z 288.723,A -85,B 0,C 180,E1 -6319.89,E2 -6319.89} C_VEL
LIN {X 0,Y 495.764,Z 288.734,A -85,B 0,C 180,E1 -6322.86,E2 -6322.86} C_VEL
LIN {X 0,Y 495.795,Z 288.721,A -85,B 0,C 180,E1 -6326.067,E2 -6326.067} C_VEL
LIN {X 0,Y 495.776,Z 288.729,A -85,B 0,C 180,E1 -6328.814,E2 -6328.814} C_VEL
LIN {X 0,Y 495.759,Z 288.727,A -85,B 0,C 180,E1 -6331.725,E2 -6331.725} C_VEL
LIN {X 0,Y 495.772,Z 288.726,A -85,B 0,C 180,E1 -6334.693,E2 -6334.693} C_VEL
LIN {X 0,Y 495.725,Z 288.735,A -85,B 0,C 180,E1 -6337.562,E2 -6337.562} C_VEL
LIN {X 0,Y 495.77,Z 288.724,A -85,B 0,C 180,E1 -6340.699,E2 -6340.699} C_VEL
LIN {X 0,Y 495.732,Z 288.732,A -85,B 0,C 180,E1 -6344.001,E2 -6344.001} C_VEL
LIN {X 0,Y 495.729,Z 288.731,A -85,B 0,C 180,E1 -6347.116,E2 -6347.116} C_VEL
LIN {X 0,Y 495.762,Z 288.731,A -85,B 0,C 180,E1 -6349.952,E2 -6349.952} C_VEL
LIN {X 0,Y 495.731,Z 288.729,A -85,B 0,C 180,E1 -6352.553,E2 -6352.553} C_VEL
LIN {X 0,Y 495.781,Z 288.725,A -85,B 0,C 180,E1 -6355.456,E2 -6355.456} C_VEL
LIN {X 0,Y 495.759,Z 288.73,A -85,B 0,C 180,E1 -6358.363,E2 -6358.363} C_VEL
LIN {X 0,Y 495.757,Z 288.727,A -85,B 0,C 180,E1 -6360.749,E2 -6360.749} C_VEL
LIN {X 0,Y 495.099,Z 288.809,A -85,B 0,C 180,E1 -6361.428,E2 -6361.428} C_VEL
LIN {X 0,Y 492.242,Z 289.167,A -85,B 0,C 180,E1 -6362.531,E2 -6362.531} C_VEL
LIN {X 0,Y 489.828,Z 289.466,A -85,B 0,C 180,E1 -6363.42,E2 -6363.42} C_VEL
LIN {X 0,Y 488.804,Z 289.6,A -85,B 0,C 180,E1 -6364.106,E2 -6364.106} C_VEL
LIN {X 0,Y 488.727,Z 289.606,A -85,B 0,C 180,E1 -6364.338,E2 -6364.338} C_VEL
LIN {X 0,Y 488.725,Z 289.602,A -85,B 0,C 180,E1 -6367.152,E2 -6367.152} C_VEL
LIN {X 0,Y 488.728,Z 289.603,A -85,B 0,C 180,E1 -6369.81,E2 -6369.81} C_VEL
LIN {X 0,Y 488.732,Z 289.609,A -85,B 0,C 180,E1 -6372.422,E2 -6372.422} C_VEL
LIN {X 0,Y 488.764,Z 289.6,A -85,B 0,C 180,E1 -6374.999,E2 -6374.999} C_VEL
LIN {X 0,Y 488.808,Z 289.596,A -85,B 0,C 180,E1 -6378.387,E2 -6378.387} C_VEL
LIN {X 0,Y 488.787,Z 289.597,A -85,B 0,C 180,E1 -6381.732,E2 -6381.732} C_VEL
LIN {X 0,Y 488.881,Z 289.592,A -85,B 0,C 180,E1 -6384.689,E2 -6384.689} C_VEL
LIN {X 0,Y 489.56,Z 296.356,A -85,B 0,C 180,E1 -6386.089,E2 -6386.089} C_VEL
LIN {X 0,Y 489.284,Z 310.237,A -85,B 0,C 180,E1 -6388.797,E2 -6388.797} C_VEL
LIN {X 0,Y 491.766,Z 323.185,A -85,B 0,C 180,E1 -6389.078,E2 -6389.078} C_VEL
LIN {X 0,Y 491.09,Z 417.547,A -85,B 0,C 180,E1 -6390.486,E2 -6390.486} C_VEL
LIN {X 0,Y 490.856,Z 430.565,A -85,B 0,C 180,E1 -6390.845,E2 -6390.845} C_VEL
LIN {X 0,Y 490.593,Z 443.631,A -85,B 0,C 180,E1 -6391.384,E2 -6391.384} C_VEL
LIN {X 0,Y 490.237,Z 455.462,A -85,B 0,C 180,E1 -6392.053,E2 -6392.053} C_VEL
LIN {X 0,Y 489.794,Z 466.823,A -85,B 0,C 180,E1 -6392.877,E2 -6392.877} C_VEL
LIN {X 0,Y 489.36,Z 477.082,A -85,B 0,C 180,E1 -6393.807,E2 -6393.807} C_VEL
LIN {X 0,Y 489.028,Z 485.475,A -85,B 0,C 180,E1 -6394.739,E2 -6394.739} C_VEL
LIN {X 0,Y 488.654,Z 494.592,A -85,B 0,C 180,E1 -6395.984,E2 -6395.984} C_VEL
LIN {X 0,Y 488.474,Z 501.741,A -85,B 0,C 180,E1 -6397.196,E2 -6397.196} C_VEL
LIN {X 0,Y 488.253,Z 506.94,A -85,B 0,C 180,E1 -6398.275,E2 -6398.275} C_VEL
LIN {X 0,Y 488.087,Z 511.805,A -85,B 0,C 180,E1 -6399.53,E2 -6399.53} C_VEL
LIN {X 0,Y 488.012,Z 515.547,A -85,B 0,C 180,E1 -6400.789,E2 -6400.789} C_VEL
LIN {X 0,Y 487.996,Z 517.571,A -85,B 0,C 180,E1 -6401.673,E2 -6401.673} C_VEL
LIN {X 0,Y 487.859,Z 518.974,A -85,B 0,C 180,E1 -6402.478,E2 -6402.478} C_VEL
LIN {X 0,Y 487.851,Z 520.013,A -85,B 0,C 180,E1 -6403.325,E2 -6403.325} C_VEL
LIN {X 0,Y 487.849,Z 520.656,A -85,B 0,C 180,E1 -6404.175,E2 -6404.175} C_VEL
LIN {X 0,Y 487.876,Z 520.88,A -85,B 0,C 180,E1 -6405.17,E2 -6405.17} C_VEL
LIN {X 0,Y 487.797,Z 520.047,A -85,B 0,C 180,E1 -6406.746,E2 -6406.746} C_VEL
LIN {X 0,Y 487.892,Z 518.243,A -85,B 0,C 180,E1 -6408.063,E2 -6408.063} C_VEL
LIN {X 0,Y 487.993,Z 515.479,A -85,B 0,C 180,E1 -6409.343,E2 -6409.343} C_VEL
LIN {X 0,Y 488.106,Z 511.634,A -85,B 0,C 180,E1 -6410.626,E2 -6410.626} C_VEL
LIN {X 0,Y 488.241,Z 506.316,A -85,B 0,C 180,E1 -6411.977,E2 -6411.977} C_VEL
LIN {X 0,Y 488.497,Z 499.85,A -85,B 0,C 180,E1 -6413.263,E2 -6413.263} C_VEL
LIN {X 0,Y 488.807,Z 492.641,A -85,B 0,C 180,E1 -6414.415,E2 -6414.415} C_VEL
LIN {X 0,Y 489.141,Z 484.081,A -85,B 0,C 180,E1 -6415.532,E2 -6415.532} C_VEL
LIN {X 0,Y 489.531,Z 474.717,A -85,B 0,C 180,E1 -6416.531,E2 -6416.531} C_VEL
LIN {X 0,Y 489.914,Z 464.246,A -85,B 0,C 180,E1 -6417.44,E2 -6417.44} C_VEL
LIN {X 0,Y 490.357,Z 452.745,A -85,B 0,C 180,E1 -6418.225,E2 -6418.225} C_VEL
LIN {X 0,Y 490.693,Z 441.008,A -85,B 0,C 180,E1 -6418.847,E2 -6418.847} C_VEL
LIN {X 0,Y 491.021,Z 427.876,A -85,B 0,C 180,E1 -6419.353,E2 -6419.353} C_VEL
LIN {X 0,Y 491.218,Z 415.265,A -85,B 0,C 180,E1 -6419.664,E2 -6419.664} C_VEL
LIN {X 0,Y 491.852,Z 323.503,A -85,B 0,C 180,E1 -6421.028,E2 -6421.028} C_VEL
LIN {X 0,Y 489.311,Z 310.111,A -85,B 0,C 180,E1 -6421.333,E2 -6421.333} C_VEL
LIN {X 0,Y 489.504,Z 294.334,A -85,B 0,C 180,E1 -6424.298,E2 -6424.298} C_VEL
LIN {X 0,Y 488.677,Z 289.618,A -85,B 0,C 180,E1 -6425.242,E2 -6425.242} C_VEL
LIN {X 0,Y 488.641,Z 289.617,A -85,B 0,C 180,E1 -6428.201,E2 -6428.201} C_VEL
LIN {X 0,Y 488.683,Z 289.611,A -85,B 0,C 180,E1 -6430.34,E2 -6430.34} C_VEL
LIN {X 0,Y 488.652,Z 289.618,A -85,B 0,C 180,E1 -6433.656,E2 -6433.656} C_VEL
LIN {X 0,Y 488.662,Z 289.608,A -85,B 0,C 180,E1 -6436.343,E2 -6436.343} C_VEL
LIN {X 0,Y 488.691,Z 289.615,A -85,B 0,C 180,E1 -6439.673,E2 -6439.673} C_VEL
LIN {X 0,Y 488.645,Z 289.614,A -85,B 0,C 180,E1 -6442.838,E2 -6442.838} C_VEL
LIN {X 0,Y 488.708,Z 289.611,A -85,B 0,C 180,E1 -6445.886,E2 -6445.886} C_VEL
LIN {X 0,Y 488.678,Z 289.607,A -85,B 0,C 180,E1 -6448.819,E2 -6448.819} C_VEL
LIN {X 0,Y 488.697,Z 289.612,A -85,B 0,C 180,E1 -6451.668,E2 -6451.668} C_VEL
LIN {X 0,Y 488.687,Z 289.607,A -85,B 0,C 180,E1 -6454.441,E2 -6454.441} C_VEL
LIN {X 0,Y 488.707,Z 289.605,A -85,B 0,C 180,E1 -6457.153,E2 -6457.153} C_VEL
LIN {X 0,Y 488.709,Z 289.607,A -85,B 0,C 180,E1 -6459.81,E2 -6459.81} C_VEL
LIN {X 0,Y 488.696,Z 289.607,A -85,B 0,C 180,E1 -6462.422,E2 -6462.422} C_VEL
LIN {X 0,Y 488.742,Z 289.6,A -85,B 0,C 180,E1 -6464.999,E2 -6464.999} C_VEL
LIN {X 0,Y 488.79,Z 289.598,A -85,B 0,C 180,E1 -6468.387,E2 -6468.387} C_VEL
LIN {X 0,Y 488.802,Z 289.594,A -85,B 0,C 180,E1 -6471.734,E2 -6471.734} C_VEL
LIN {X 0,Y 488.789,Z 289.595,A -85,B 0,C 180,E1 -6475.051,E2 -6475.051} C_VEL
LIN {X 0,Y 488.944,Z 289.572,A -85,B 0,C 180,E1 -6477.529,E2 -6477.529} C_VEL
LIN {X 0,Y 488.962,Z 289.577,A -85,B 0,C 180,E1 -6480.824,E2 -6480.824} C_VEL
LIN {X 0,Y 488.945,Z 289.579,A -85,B 0,C 180,E1 -6482.472,E2 -6482.472} C_VEL
LIN {X 0,Y 488.834,Z 289.588,A -85,B 0,C 180,E1 -6485.776,E2 -6485.776} C_VEL
LIN {X 0,Y 488.804,Z 289.593,A -85,B 0,C 180,E1 -6488.267,E2 -6488.267} C_VEL
LIN {X 0,Y 488.794,Z 289.593,A -85,B 0,C 180,E1 -6491.613,E2 -6491.613} C_VEL
LIN {X 0,Y 488.748,Z 289.606,A -85,B 0,C 180,E1 -6495.001,E2 -6495.001} C_VEL
LIN {X 0,Y 488.741,Z 289.601,A -85,B 0,C 180,E1 -6498.443,E2 -6498.443} C_VEL
LIN {X 0,Y 488.695,Z 289.614,A -85,B 0,C 180,E1 -6501.071,E2 -6501.071} C_VEL
LIN {X 0,Y 488.681,Z 289.606,A -85,B 0,C 180,E1 -6503.746,E2 -6503.746} C_VEL
LIN {X 0,Y 488.787,Z 289.601,A -85,B 0,C 180,E1 -6506.946,E2 -6506.946} C_VEL
LIN {X 0,Y 488.708,Z 289.605,A -85,B 0,C 180,E1 -6510.366,E2 -6510.366} C_VEL
LIN {X 0,Y 488.725,Z 289.61,A -85,B 0,C 180,E1 -6513.486,E2 -6513.486} C_VEL
LIN {X 0,Y 488.68,Z 289.608,A -85,B 0,C 180,E1 -6516.357,E2 -6516.357} C_VEL
LIN {X 0,Y 488.735,Z 289.608,A -85,B 0,C 180,E1 -6519.251,E2 -6519.251} C_VEL
LIN {X 0,Y 488.686,Z 289.607,A -85,B 0,C 180,E1 -6522.526,E2 -6522.526} C_VEL
LIN {X 0,Y 488.704,Z 289.608,A -85,B 0,C 180,E1 -6525.2,E2 -6525.2} C_VEL
LIN {X 0,Y 488.724,Z 289.607,A -85,B 0,C 180,E1 -6527.48,E2 -6527.48} C_VEL
LIN {X 0,Y 488.736,Z 289.6,A -85,B 0,C 180,E1 -6530.751,E2 -6530.751} C_VEL
LIN {X 0,Y 488.679,Z 289.613,A -85,B 0,C 180,E1 -6533.87,E2 -6533.87} C_VEL
LIN {X 0,Y 488.733,Z 289.602,A -85,B 0,C 180,E1 -6536.879,E2 -6536.879} C_VEL
LIN {X 0,Y 488.72,Z 289.611,A -85,B 0,C 180,E1 -6539.782,E2 -6539.782} C_VEL
LIN {X 0,Y 488.789,Z 289.599,A -85,B 0,C 180,E1 -6543.058,E2 -6543.058} C_VEL
LIN {X 0,Y 488.788,Z 289.687,A -85,B 0,C 180,E1 -6544.548,E2 -6544.548} C_VEL
LIN {X 0,Y 490.686,Z 300.182,A -85,B 0,C 180,E1 -6546.443,E2 -6546.443} C_VEL
LIN {X 0,Y 490.127,Z 316.763,A -85,B 0,C 180,E1 -6549.215,E2 -6549.215} C_VEL
LIN {X 0,Y 489.505,Z 335.152,A -85,B 0,C 180,E1 -6552.238,E2 -6552.238} C_VEL
LIN {X 0,Y 489.248,Z 344.305,A -85,B 0,C 180,E1 -6553.715,E2 -6553.715} C_VEL
LIN {X 0,Y 491.677,Z 360.691,A -85,B 0,C 180,E1 -6554.046,E2 -6554.046} C_VEL
LIN {X 0,Y 491.097,Z 452.643,A -85,B 0,C 180,E1 -6555.419,E2 -6555.419} C_VEL
LIN {X 0,Y 490.76,Z 465.915,A -85,B 0,C 180,E1 -6555.779,E2 -6555.779} C_VEL
LIN {X 0,Y 490.38,Z 479.213,A -85,B 0,C 180,E1 -6556.323,E2 -6556.323} C_VEL
LIN {X 0,Y 490.025,Z 490.667,A -85,B 0,C 180,E1 -6556.965,E2 -6556.965} C_VEL
LIN {X 0,Y 489.548,Z 502,A -85,B 0,C 180,E1 -6557.776,E2 -6557.776} C_VEL
LIN {X 0,Y 489.169,Z 512.466,A -85,B 0,C 180,E1 -6558.713,E2 -6558.713} C_VEL
LIN {X 0,Y 488.834,Z 521.026,A -85,B 0,C 180,E1 -6559.648,E2 -6559.648} C_VEL
LIN {X 0,Y 488.519,Z 528.928,A -85,B 0,C 180,E1 -6560.687,E2 -6560.687} C_VEL
LIN {X 0,Y 488.275,Z 536.649,A -85,B 0,C 180,E1 -6561.934,E2 -6561.934} C_VEL
LIN {X 0,Y 488.1,Z 543.771,A -85,B 0,C 180,E1 -6563.387,E2 -6563.387} C_VEL
LIN {X 0,Y 488.017,Z 548.513,A -85,B 0,C 180,E1 -6564.63,E2 -6564.63} C_VEL
LIN {X 0,Y 487.928,Z 552.136,A -85,B 0,C 180,E1 -6565.871,E2 -6565.871} C_VEL
LIN {X 0,Y 487.964,Z 554.009,A -85,B 0,C 180,E1 -6566.699,E2 -6566.699} C_VEL
LIN {X 0,Y 487.89,Z 556.412,A -85,B 0,C 180,E1 -6568.35,E2 -6568.35} C_VEL
LIN {X 0,Y 487.822,Z 557.242,A -85,B 0,C 180,E1 -6570.001,E2 -6570.001} C_VEL
LIN {X 0,Y 487.891,Z 556.422,A -85,B 0,C 180,E1 -6571.652,E2 -6571.652} C_VEL
LIN {X 0,Y 487.909,Z 555.427,A -85,B 0,C 180,E1 -6572.478,E2 -6572.478} C_VEL
LIN {X 0,Y 487.965,Z 554.029,A -85,B 0,C 180,E1 -6573.304,E2 -6573.304} C_VEL
LIN {X 0,Y 487.921,Z 551.085,A -85,B 0,C 180,E1 -6574.545,E2 -6574.545} C_VEL
LIN {X 0,Y 488.023,Z 547.102,A -85,B 0,C 180,E1 -6575.787,E2 -6575.787} C_VEL
LIN {X 0,Y 488.183,Z 540.974,A -85,B 0,C 180,E1 -6577.238,E2 -6577.238} C_VEL
LIN {X 0,Y 488.359,Z 534.274,A -85,B 0,C 180,E1 -6578.484,E2 -6578.484} C_VEL
LIN {X 0,Y 488.648,Z 525.961,A -85,B 0,C 180,E1 -6579.73,E2 -6579.73} C_VEL
LIN {X 0,Y 488.979,Z 517.433,A -85,B 0,C 180,E1 -6580.77,E2 -6580.77} C_VEL
LIN {X 0,Y 489.457,Z 506.9,A -85,B 0,C 180,E1 -6581.808,E2 -6581.808} C_VEL
LIN {X 0,Y 489.817,Z 495.184,A -85,B 0,C 180,E1 -6582.735,E2 -6582.735} C_VEL
LIN {X 0,Y 490.232,Z 483.075,A -85,B 0,C 180,E1 -6583.473,E2 -6583.473} C_VEL
LIN {X 0,Y 490.628,Z 470.629,A -85,B 0,C 180,E1 -6584.042,E2 -6584.042} C_VEL
LIN {X 0,Y 490.978,Z 457.773,A -85,B 0,C 180,E1 -6584.455,E2 -6584.455} C_VEL
LIN {X 0,Y 491.132,Z 444.095,A -85,B 0,C 180,E1 -6584.715,E2 -6584.715} C_VEL
LIN {X 0,Y 491.578,Z 359.729,A -85,B 0,C 180,E1 -6585.958,E2 -6585.958} C_VEL
LIN {X 0,Y 489.262,Z 344.373,A -85,B 0,C 180,E1 -6586.268,E2 -6586.268} C_VEL
LIN {X 0,Y 489.892,Z 324.704,A -85,B 0,C 180,E1 -6589.485,E2 -6589.485} C_VEL
LIN {X 0,Y 490.575,Z 304.963,A -85,B 0,C 180,E1 -6592.757,E2 -6592.757} C_VEL
LIN {X 0,Y 490.65,Z 299.675,A -85,B 0,C 180,E1 -6593.646,E2 -6593.646} C_VEL
LIN {X 0,Y 488.798,Z 289.6,A -85,B 0,C 180,E1 -6595.456,E2 -6595.456} C_VEL
LIN {X 0,Y 488.748,Z 289.606,A -85,B 0,C 180,E1 -6598.33,E2 -6598.33} C_VEL
LIN {X 0,Y 488.698,Z 289.605,A -85,B 0,C 180,E1 -6601.18,E2 -6601.18} C_VEL
LIN {X 0,Y 488.73,Z 289.608,A -85,B 0,C 180,E1 -6604.114,E2 -6604.114} C_VEL
LIN {X 0,Y 488.685,Z 289.607,A -85,B 0,C 180,E1 -6607.159,E2 -6607.159} C_VEL
LIN {X 0,Y 488.724,Z 289.609,A -85,B 0,C 180,E1 -6610.345,E2 -6610.345} C_VEL
LIN {X 0,Y 488.69,Z 289.606,A -85,B 0,C 180,E1 -6613.655,E2 -6613.655} C_VEL
LIN {X 0,Y 488.69,Z 289.61,A -85,B 0,C 180,E1 -6616.346,E2 -6616.346} C_VEL
LIN {X 0,Y 488.739,Z 289.6,A -85,B 0,C 180,E1 -6619.677,E2 -6619.677} C_VEL
LIN {X 0,Y 488.685,Z 289.616,A -85,B 0,C 180,E1 -6622.841,E2 -6622.841} C_VEL
LIN {X 0,Y 488.726,Z 289.601,A -85,B 0,C 180,E1 -6625.887,E2 -6625.887} C_VEL
LIN {X 0,Y 488.698,Z 289.61,A -85,B 0,C 180,E1 -6628.82,E2 -6628.82} C_VEL
LIN {X 0,Y 488.749,Z 289.601,A -85,B 0,C 180,E1 -6631.671,E2 -6631.671} C_VEL
LIN {X 0,Y 488.745,Z 289.599,A -85,B 0,C 180,E1 -6634.444,E2 -6634.444} C_VEL
LIN {X 0,Y 488.728,Z 289.607,A -85,B 0,C 180,E1 -6637.153,E2 -6637.153} C_VEL
LIN {X 0,Y 488.73,Z 289.605,A -85,B 0,C 180,E1 -6639.81,E2 -6639.81} C_VEL
LIN {X 0,Y 488.719,Z 289.602,A -85,B 0,C 180,E1 -6642.423,E2 -6642.423} C_VEL
LIN {X 0,Y 488.767,Z 289.598,A -85,B 0,C 180,E1 -6645,E2 -6645} C_VEL
LIN {X 0,Y 488.811,Z 289.592,A -85,B 0,C 180,E1 -6648.387,E2 -6648.387} C_VEL
LIN {X 0,Y 488.82,Z 289.598,A -85,B 0,C 180,E1 -6651.733,E2 -6651.733} C_VEL
LIN {X 0,Y 488.809,Z 289.591,A -85,B 0,C 180,E1 -6655.051,E2 -6655.051} C_VEL
LIN {X 0,Y 488.965,Z 289.574,A -85,B 0,C 180,E1 -6657.528,E2 -6657.528} C_VEL
LIN {X 0,Y 488.919,Z 289.578,A -85,B 0,C 180,E1 -6660.823,E2 -6660.823} C_VEL
LIN {X 0,Y 488.963,Z 289.577,A -85,B 0,C 180,E1 -6662.471,E2 -6662.471} C_VEL
LIN {X 0,Y 488.85,Z 289.588,A -85,B 0,C 180,E1 -6665.776,E2 -6665.776} C_VEL
LIN {X 0,Y 488.79,Z 289.601,A -85,B 0,C 180,E1 -6668.267,E2 -6668.267} C_VEL
LIN {X 0,Y 488.81,Z 289.591,A -85,B 0,C 180,E1 -6671.612,E2 -6671.612} C_VEL
LIN {X 0,Y 488.769,Z 289.599,A -85,B 0,C 180,E1 -6675,E2 -6675} C_VEL
LIN {X 0,Y 488.752,Z 289.603,A -85,B 0,C 180,E1 -6678.442,E2 -6678.442} C_VEL
LIN {X 0,Y 488.711,Z 289.608,A -85,B 0,C 180,E1 -6681.07,E2 -6681.07} C_VEL
LIN {X 0,Y 488.692,Z 289.606,A -85,B 0,C 180,E1 -6683.745,E2 -6683.745} C_VEL
LIN {X 0,Y 488.797,Z 289.602,A -85,B 0,C 180,E1 -6686.943,E2 -6686.943} C_VEL
LIN {X 0,Y 488.714,Z 289.603,A -85,B 0,C 180,E1 -6690.362,E2 -6690.362} C_VEL
LIN {X 0,Y 488.738,Z 289.605,A -85,B 0,C 180,E1 -6693.484,E2 -6693.484} C_VEL
LIN {X 0,Y 488.677,Z 289.607,A -85,B 0,C 180,E1 -6696.352,E2 -6696.352} C_VEL
LIN {X 0,Y 488.705,Z 289.611,A -85,B 0,C 180,E1 -6699.254,E2 -6699.254} C_VEL
LIN {X 0,Y 488.711,Z 289.611,A -85,B 0,C 180,E1 -6701.599,E2 -6701.599} C_VEL
LIN {X 0,Y 488.705,Z 289.604,A -85,B 0,C 180,E1 -6704.802,E2 -6704.802} C_VEL
LIN {X 0,Y 488.695,Z 289.612,A -85,B 0,C 180,E1 -6707.474,E2 -6707.474} C_VEL
LIN {X 0,Y 488.737,Z 289.609,A -85,B 0,C 180,E1 -6709.676,E2 -6709.676} C_VEL
LIN {X 0,Y 488.682,Z 289.607,A -85,B 0,C 180,E1 -6712.84,E2 -6712.84} C_VEL
LIN {X 0,Y 488.734,Z 289.609,A -85,B 0,C 180,E1 -6715.886,E2 -6715.886} C_VEL
LIN {X 0,Y 488.695,Z 289.606,A -85,B 0,C 180,E1 -6718.819,E2 -6718.819} C_VEL
LIN {X 0,Y 488.749,Z 289.601,A -85,B 0,C 180,E1 -6721.671,E2 -6721.671} C_VEL
LIN {X 0,Y 488.727,Z 289.606,A -85,B 0,C 180,E1 -6724.338,E2 -6724.338} C_VEL
LIN {X 0,Y 488.076,Z 289.692,A -85,B 0,C 180,E1 -6725.026,E2 -6725.026} C_VEL
LIN {X 0,Y 485.214,Z 290.047,A -85,B 0,C 180,E1 -6726.143,E2 -6726.143} C_VEL
LIN {X 0,Y 482.779,Z 290.346,A -85,B 0,C 180,E1 -6727.043,E2 -6727.043} C_VEL
LIN {X 0,Y 481.727,Z 290.475,A -85,B 0,C 180,E1 -6727.738,E2 -6727.738} C_VEL
LIN {X 0,Y 481.639,Z 290.485,A -85,B 0,C 180,E1 -6727.974,E2 -6727.974} C_VEL
LIN {X 0,Y 481.709,Z 290.485,A -85,B 0,C 180,E1 -6730.392,E2 -6730.392} C_VEL
LIN {X 0,Y 481.69,Z 290.48,A -85,B 0,C 180,E1 -6733.033,E2 -6733.033} C_VEL
LIN {X 0,Y 481.691,Z 290.478,A -85,B 0,C 180,E1 -6735.638,E2 -6735.638} C_VEL
LIN {X 0,Y 481.753,Z 290.473,A -85,B 0,C 180,E1 -6738.214,E2 -6738.214} C_VEL
LIN {X 0,Y 481.741,Z 290.475,A -85,B 0,C 180,E1 -6741.61,E2 -6741.61} C_VEL
LIN {X 0,Y 481.858,Z 290.614,A -85,B 0,C 180,E1 -6744.611,E2 -6744.611} C_VEL
LIN {X 0,Y 482.645,Z 296.522,A -85,B 0,C 180,E1 -6745.824,E2 -6745.824} C_VEL
LIN {X 0,Y 482.31,Z 310.452,A -85,B 0,C 180,E1 -6748.566,E2 -6748.566} C_VEL
LIN {X 0,Y 484.981,Z 324.89,A -85,B 0,C 180,E1 -6748.881,E2 -6748.881} C_VEL
LIN {X 0,Y 484.214,Z 417.859,A -85,B 0,C 180,E1 -6750.285,E2 -6750.285} C_VEL
LIN {X 0,Y 483.967,Z 430.872,A -85,B 0,C 180,E1 -6750.649,E2 -6750.649} C_VEL
LIN {X 0,Y 483.711,Z 443.926,A -85,B 0,C 180,E1 -6751.196,E2 -6751.196} C_VEL
LIN {X 0,Y 483.332,Z 455.763,A -85,B 0,C 180,E1 -6751.874,E2 -6751.874} C_VEL
LIN {X 0,Y 482.841,Z 467.141,A -85,B 0,C 180,E1 -6752.71,E2 -6752.71} C_VEL
LIN {X 0,Y 482.383,Z 477.393,A -85,B 0,C 180,E1 -6753.653,E2 -6753.653} C_VEL
LIN {X 0,Y 482.041,Z 485.774,A -85,B 0,C 180,E1 -6754.598,E2 -6754.598} C_VEL
LIN {X 0,Y 481.631,Z 494.886,A -85,B 0,C 180,E1 -6755.861,E2 -6755.861} C_VEL
LIN {X 0,Y 481.453,Z 501.348,A -85,B 0,C 180,E1 -6756.962,E2 -6756.962} C_VEL
LIN {X 0,Y 481.171,Z 508.13,A -85,B 0,C 180,E1 -6758.397,E2 -6758.397} C_VEL
LIN {X 0,Y 480.992,Z 512.803,A -85,B 0,C 180,E1 -6759.672,E2 -6759.672} C_VEL
LIN {X 0,Y 480.914,Z 516.363,A -85,B 0,C 180,E1 -6760.95,E2 -6760.95} C_VEL
LIN {X 0,Y 480.886,Z 518.165,A -85,B 0,C 180,E1 -6761.805,E2 -6761.805} C_VEL
LIN {X 0,Y 480.773,Z 519.53,A -85,B 0,C 180,E1 -6762.665,E2 -6762.665} C_VEL
LIN {X 0,Y 480.749,Z 520.488,A -85,B 0,C 180,E1 -6763.525,E2 -6763.525} C_VEL
LIN {X 0,Y 480.762,Z 521.037,A -85,B 0,C 180,E1 -6764.388,E2 -6764.388} C_VEL
LIN {X 0,Y 480.785,Z 521.13,A -85,B 0,C 180,E1 -6765.254,E2 -6765.254} C_VEL
LIN {X 0,Y 480.698,Z 520.82,A -85,B 0,C 180,E1 -6766.127,E2 -6766.127} C_VEL
LIN {X 0,Y 480.711,Z 520.1,A -85,B 0,C 180,E1 -6767,E2 -6767} C_VEL
LIN {X 0,Y 480.817,Z 518.393,A -85,B 0,C 180,E1 -6768.179,E2 -6768.179} C_VEL
LIN {X 0,Y 480.938,Z 515.173,A -85,B 0,C 180,E1 -6769.638,E2 -6769.638} C_VEL
LIN {X 0,Y 481.061,Z 510.754,A -85,B 0,C 180,E1 -6771.045,E2 -6771.045} C_VEL
LIN {X 0,Y 481.234,Z 505.542,A -85,B 0,C 180,E1 -6772.314,E2 -6772.314} C_VEL
LIN {X 0,Y 481.543,Z 498.531,A -85,B 0,C 180,E1 -6773.661,E2 -6773.661} C_VEL
LIN {X 0,Y 481.861,Z 491.27,A -85,B 0,C 180,E1 -6774.79,E2 -6774.79} C_VEL
LIN {X 0,Y 482.252,Z 482.392,A -85,B 0,C 180,E1 -6775.924,E2 -6775.924} C_VEL
LIN {X 0,Y 482.66,Z 473.706,A -85,B 0,C 180,E1 -6776.831,E2 -6776.831} C_VEL
LIN {X 0,Y 483.076,Z 462.974,A -85,B 0,C 180,E1 -6777.744,E2 -6777.744} C_VEL
LIN {X 0,Y 483.538,Z 451.085,A -85,B 0,C 180,E1 -6778.541,E2 -6778.541} C_VEL
LIN {X 0,Y 483.896,Z 438.796,A -85,B 0,C 180,E1 -6779.171,E2 -6779.171} C_VEL
LIN {X 0,Y 484.205,Z 425.673,A -85,B 0,C 180,E1 -6779.643,E2 -6779.643} C_VEL
LIN {X 0,Y 484.434,Z 412.343,A -85,B 0,C 180,E1 -6779.942,E2 -6779.942} C_VEL
LIN {X 0,Y 484.99,Z 323.641,A -85,B 0,C 180,E1 -6781.275,E2 -6781.275} C_VEL
LIN {X 0,Y 482.351,Z 310.314,A -85,B 0,C 180,E1 -6781.593,E2 -6781.593} C_VEL
LIN {X 0,Y 482.548,Z 295.546,A -85,B 0,C 180,E1 -6784.402,E2 -6784.402} C_VEL
LIN {X 0,Y 481.646,Z 290.493,A -85,B 0,C 180,E1 -6785.42,E2 -6785.42} C_VEL
LIN {X 0,Y 481.617,Z 290.494,A -85,B 0,C 180,E1 -6788.862,E2 -6788.862} C_VEL
LIN {X 0,Y 481.609,Z 290.493,A -85,B 0,C 180,E1 -6791.907,E2 -6791.907} C_VEL
LIN {X 0,Y 481.638,Z 290.487,A -85,B 0,C 180,E1 -6794.457,E2 -6794.457} C_VEL
LIN {X 0,Y 481.608,Z 290.488,A -85,B 0,C 180,E1 -6796.854,E2 -6796.854} C_VEL
LIN {X 0,Y 481.642,Z 290.488,A -85,B 0,C 180,E1 -6800.056,E2 -6800.056} C_VEL
LIN {X 0,Y 481.603,Z 290.495,A -85,B 0,C 180,E1 -6803.377,E2 -6803.377} C_VEL
LIN {X 0,Y 481.662,Z 290.485,A -85,B 0,C 180,E1 -6806.326,E2 -6806.326} C_VEL
LIN {X 0,Y 481.636,Z 290.488,A -85,B 0,C 180,E1 -6809.417,E2 -6809.417} C_VEL
LIN {X 0,Y 481.651,Z 290.488,A -85,B 0,C 180,E1 -6812.165,E2 -6812.165} C_VEL
LIN {X 0,Y 481.664,Z 290.48,A -85,B 0,C 180,E1 -6814.967,E2 -6814.967} C_VEL
LIN {X 0,Y 481.633,Z 290.492,A -85,B 0,C 180,E1 -6817.704,E2 -6817.704} C_VEL
LIN {X 0,Y 481.689,Z 290.483,A -85,B 0,C 180,E1 -6820.393,E2 -6820.393} C_VEL
LIN {X 0,Y 481.66,Z 290.479,A -85,B 0,C 180,E1 -6823.033,E2 -6823.033} C_VEL
LIN {X 0,Y 481.668,Z 290.484,A -85,B 0,C 180,E1 -6825.638,E2 -6825.638} C_VEL
LIN {X 0,Y 481.735,Z 290.476,A -85,B 0,C 180,E1 -6828.215,E2 -6828.215} C_VEL
LIN {X 0,Y 481.747,Z 290.472,A -85,B 0,C 180,E1 -6831.612,E2 -6831.612} C_VEL
LIN {X 0,Y 481.759,Z 290.472,A -85,B 0,C 180,E1 -6834.979,E2 -6834.979} C_VEL
LIN {X 0,Y 481.911,Z 290.448,A -85,B 0,C 180,E1 -6837.493,E2 -6837.493} C_VEL
LIN {X 0,Y 481.911,Z 290.455,A -85,B 0,C 180,E1 -6840.836,E2 -6840.836} C_VEL
LIN {X 0,Y 481.913,Z 290.454,A -85,B 0,C 180,E1 -6842.508,E2 -6842.508} C_VEL
LIN {X 0,Y 481.794,Z 290.466,A -85,B 0,C 180,E1 -6845.861,E2 -6845.861} C_VEL
LIN {X 0,Y 481.749,Z 290.473,A -85,B 0,C 180,E1 -6848.389,E2 -6848.389} C_VEL
LIN {X 0,Y 481.739,Z 290.472,A -85,B 0,C 180,E1 -6851.785,E2 -6851.785} C_VEL
LIN {X 0,Y 481.728,Z 290.478,A -85,B 0,C 180,E1 -6855.225,E2 -6855.225} C_VEL
LIN {X 0,Y 481.699,Z 290.48,A -85,B 0,C 180,E1 -6858.722,E2 -6858.722} C_VEL
LIN {X 0,Y 481.634,Z 290.489,A -85,B 0,C 180,E1 -6861.395,E2 -6861.395} C_VEL
LIN {X 0,Y 481.665,Z 290.479,A -85,B 0,C 180,E1 -6864.114,E2 -6864.114} C_VEL
LIN {X 0,Y 481.74,Z 290.478,A -85,B 0,C 180,E1 -6867.142,E2 -6867.142} C_VEL
LIN {X 0,Y 481.676,Z 290.483,A -85,B 0,C 180,E1 -6869.742,E2 -6869.742} C_VEL
LIN {X 0,Y 481.662,Z 290.481,A -85,B 0,C 180,E1 -6872.675,E2 -6872.675} C_VEL
LIN {X 0,Y 481.633,Z 290.49,A -85,B 0,C 180,E1 -6875.71,E2 -6875.71} C_VEL
LIN {X 0,Y 481.706,Z 290.483,A -85,B 0,C 180,E1 -6879.355,E2 -6879.355} C_VEL
LIN {X 0,Y 481.645,Z 290.485,A -85,B 0,C 180,E1 -6882.161,E2 -6882.161} C_VEL
LIN {X 0,Y 481.652,Z 290.485,A -85,B 0,C 180,E1 -6885.544,E2 -6885.544} C_VEL
LIN {X 0,Y 481.667,Z 290.486,A -85,B 0,C 180,E1 -6888.086,E2 -6888.086} C_VEL
LIN {X 0,Y 481.691,Z 290.48,A -85,B 0,C 180,E1 -6891.145,E2 -6891.145} C_VEL
LIN {X 0,Y 481.662,Z 290.485,A -85,B 0,C 180,E1 -6894.796,E2 -6894.796} C_VEL
LIN {X 0,Y 481.667,Z 290.484,A -85,B 0,C 180,E1 -6897.327,E2 -6897.327} C_VEL
LIN {X 0,Y 481.675,Z 290.486,A -85,B 0,C 180,E1 -6900.26,E2 -6900.26} C_VEL
LIN {X 0,Y 481.743,Z 290.477,A -85,B 0,C 180,E1 -6903.114,E2 -6903.114} C_VEL
LIN {X 0,Y 481.765,Z 290.552,A -85,B 0,C 180,E1 -6904.327,E2 -6904.327} C_VEL
LIN {X 0,Y 483.687,Z 301.064,A -85,B 0,C 180,E1 -6906.262,E2 -6906.262} C_VEL
LIN {X 0,Y 483.381,Z 312.877,A -85,B 0,C 180,E1 -6908.277,E2 -6908.277} C_VEL
LIN {X 0,Y 482.678,Z 332.331,A -85,B 0,C 180,E1 -6911.539,E2 -6911.539} C_VEL
LIN {X 0,Y 482.27,Z 344.012,A -85,B 0,C 180,E1 -6913.46,E2 -6913.46} C_VEL
LIN {X 0,Y 484.875,Z 361.149,A -85,B 0,C 180,E1 -6913.816,E2 -6913.816} C_VEL
LIN {X 0,Y 484.247,Z 452.706,A -85,B 0,C 180,E1 -6915.208,E2 -6915.208} C_VEL
LIN {X 0,Y 483.901,Z 465.846,A -85,B 0,C 180,E1 -6915.573,E2 -6915.573} C_VEL
LIN {X 0,Y 483.465,Z 479.061,A -85,B 0,C 180,E1 -6916.123,E2 -6916.123} C_VEL
LIN {X 0,Y 483.112,Z 490.184,A -85,B 0,C 180,E1 -6916.756,E2 -6916.756} C_VEL
LIN {X 0,Y 482.587,Z 501.771,A -85,B 0,C 180,E1 -6917.597,E2 -6917.597} C_VEL
LIN {X 0,Y 482.185,Z 512.23,A -85,B 0,C 180,E1 -6918.547,E2 -6918.547} C_VEL
LIN {X 0,Y 481.816,Z 520.785,A -85,B 0,C 180,E1 -6919.496,E2 -6919.496} C_VEL
LIN {X 0,Y 481.47,Z 528.682,A -85,B 0,C 180,E1 -6920.55,E2 -6920.55} C_VEL
LIN {X 0,Y 481.225,Z 536.399,A -85,B 0,C 180,E1 -6921.815,E2 -6921.815} C_VEL
LIN {X 0,Y 481.019,Z 543.518,A -85,B 0,C 180,E1 -6923.289,E2 -6923.289} C_VEL
LIN {X 0,Y 480.93,Z 548.256,A -85,B 0,C 180,E1 -6924.551,E2 -6924.551} C_VEL
LIN {X 0,Y 480.828,Z 551.876,A -85,B 0,C 180,E1 -6925.81,E2 -6925.81} C_VEL
LIN {X 0,Y 480.888,Z 553.748,A -85,B 0,C 180,E1 -6926.65,E2 -6926.65} C_VEL
LIN {X 0,Y 480.821,Z 556.15,A -85,B 0,C 180,E1 -6928.326,E2 -6928.326} C_VEL
LIN {X 0,Y 480.745,Z 556.978,A -85,B 0,C 180,E1 -6930.001,E2 -6930.001} C_VEL
LIN {X 0,Y 480.821,Z 556.157,A -85,B 0,C 180,E1 -6931.676,E2 -6931.676} C_VEL
LIN {X 0,Y 480.889,Z 553.761,A -85,B 0,C 180,E1 -6933.353,E2 -6933.353} C_VEL
LIN {X 0,Y 480.839,Z 550.812,A -85,B 0,C 180,E1 -6934.612,E2 -6934.612} C_VEL
LIN {X 0,Y 480.927,Z 546.824,A -85,B 0,C 180,E1 -6935.872,E2 -6935.872} C_VEL
LIN {X 0,Y 481.108,Z 540.686,A -85,B 0,C 180,E1 -6937.345,E2 -6937.345} C_VEL
LIN {X 0,Y 481.312,Z 533.98,A -85,B 0,C 180,E1 -6938.609,E2 -6938.609} C_VEL
LIN {X 0,Y 481.593,Z 525.659,A -85,B 0,C 180,E1 -6939.874,E2 -6939.874} C_VEL
LIN {X 0,Y 481.96,Z 517.121,A -85,B 0,C 180,E1 -6940.929,E2 -6940.929} C_VEL
LIN {X 0,Y 482.468,Z 506.595,A -85,B 0,C 180,E1 -6941.98,E2 -6941.98} C_VEL
LIN {X 0,Y 482.852,Z 495.347,A -85,B 0,C 180,E1 -6942.884,E2 -6942.884} C_VEL
LIN {X 0,Y 483.231,Z 484.671,A -85,B 0,C 180,E1 -6943.564,E2 -6943.564} C_VEL
LIN {X 0,Y 483.618,Z 472.836,A -85,B 0,C 180,E1 -6944.143,E2 -6944.143} C_VEL
LIN {X 0,Y 484.04,Z 459.185,A -85,B 0,C 180,E1 -6944.613,E2 -6944.613} C_VEL
LIN {X 0,Y 484.254,Z 445.244,A -85,B 0,C 180,E1 -6944.902,E2 -6944.902} C_VEL
LIN {X 0,Y 484.799,Z 361.221,A -85,B 0,C 180,E1 -6946.153,E2 -6946.153} C_VEL
LIN {X 0,Y 482.259,Z 344.051,A -85,B 0,C 180,E1 -6946.511,E2 -6946.511} C_VEL
LIN {X 0,Y 482.899,Z 325.686,A -85,B 0,C 180,E1 -6949.558,E2 -6949.558} C_VEL
LIN {X 0,Y 483.619,Z 305.911,A -85,B 0,C 180,E1 -6952.877,E2 -6952.877} C_VEL
LIN {X 0,Y 483.673,Z 300.881,A -85,B 0,C 180,E1 -6953.734,E2 -6953.734} C_VEL
LIN {X 0,Y 481.748,Z 290.479,A -85,B 0,C 180,E1 -6955.631,E2 -6955.631} C_VEL
LIN {X 0,Y 481.704,Z 290.485,A -85,B 0,C 180,E1 -6957.833,E2 -6957.833} C_VEL
LIN {X 0,Y 481.651,Z 290.486,A -85,B 0,C 180,E1 -6960.712,E2 -6960.712} C_VEL
LIN {X 0,Y 481.681,Z 290.481,A -85,B 0,C 180,E1 -6963.73,E2 -6963.73} C_VEL
LIN {X 0,Y 481.631,Z 290.489,A -85,B 0,C 180,E1 -6966.747,E2 -6966.747} C_VEL
LIN {X 0,Y 481.681,Z 290.481,A -85,B 0,C 180,E1 -6969.941,E2 -6969.941} C_VEL
LIN {X 0,Y 481.638,Z 290.486,A -85,B 0,C 180,E1 -6973.147,E2 -6973.147} C_VEL
LIN {X 0,Y 481.66,Z 290.482,A -85,B 0,C 180,E1 -6975.642,E2 -6975.642} C_VEL
LIN {X 0,Y 481.662,Z 290.488,A -85,B 0,C 180,E1 -6978.959,E2 -6978.959} C_VEL
LIN {X 0,Y 481.66,Z 290.482,A -85,B 0,C 180,E1 -6981.993,E2 -6981.993} C_VEL
LIN {X 0,Y 481.689,Z 290.482,A -85,B 0,C 180,E1 -6985.318,E2 -6985.318} C_VEL
LIN {X 0,Y 481.649,Z 290.484,A -85,B 0,C 180,E1 -6988.312,E2 -6988.312} C_VEL
LIN {X 0,Y 481.705,Z 290.485,A -85,B 0,C 180,E1 -6991.219,E2 -6991.219} C_VEL
LIN {X 0,Y 481.702,Z 290.477,A -85,B 0,C 180,E1 -6994.043,E2 -6994.043} C_VEL
LIN {X 0,Y 481.68,Z 290.481,A -85,B 0,C 180,E1 -6996.812,E2 -6996.812} C_VEL
LIN {X 0,Y 481.701,Z 290.485,A -85,B 0,C 180,E1 -6999.503,E2 -6999.503} C_VEL
LIN {X 0,Y 481.697,Z 290.478,A -85,B 0,C 180,E1 -7002.158,E2 -7002.158} C_VEL
LIN {X 0,Y 481.748,Z 290.471,A -85,B 0,C 180,E1 -7004.776,E2 -7004.776} C_VEL
LIN {X 0,Y 481.756,Z 290.472,A -85,B 0,C 180,E1 -7008.215,E2 -7008.215} C_VEL
LIN {X 0,Y 481.765,Z 290.474,A -85,B 0,C 180,E1 -7011.612,E2 -7011.612} C_VEL
LIN {X 0,Y 481.779,Z 290.467,A -85,B 0,C 180,E1 -7014.979,E2 -7014.979} C_VEL
LIN {X 0,Y 481.932,Z 290.45,A -85,B 0,C 180,E1 -7017.492,E2 -7017.492} C_VEL
LIN {X 0,Y 481.944,Z 290.454,A -85,B 0,C 180,E1 -7020,E2 -7020} C_VEL
LIN {X 0,Y 481.93,Z 290.452,A -85,B 0,C 180,E1 -7022.507,E2 -7022.507} C_VEL
LIN {X 0,Y 481.811,Z 290.466,A -85,B 0,C 180,E1 -7025.86,E2 -7025.86} C_VEL
LIN {X 0,Y 481.745,Z 290.481,A -85,B 0,C 180,E1 -7028.388,E2 -7028.388} C_VEL
LIN {X 0,Y 481.756,Z 290.47,A -85,B 0,C 180,E1 -7031.785,E2 -7031.785} C_VEL
LIN {X 0,Y 481.749,Z 290.472,A -85,B 0,C 180,E1 -7035.224,E2 -7035.224} C_VEL
LIN {X 0,Y 481.713,Z 290.485,A -85,B 0,C 180,E1 -7038.721,E2 -7038.721} C_VEL
LIN {X 0,Y 481.65,Z 290.484,A -85,B 0,C 180,E1 -7041.394,E2 -7041.394} C_VEL
LIN {X 0,Y 481.678,Z 290.48,A -85,B 0,C 180,E1 -7044.113,E2 -7044.113} C_VEL
LIN {X 0,Y 481.751,Z 290.477,A -85,B 0,C 180,E1 -7047.139,E2 -7047.139} C_VEL
LIN {X 0,Y 481.683,Z 290.48,A -85,B 0,C 180,E1 -7049.741,E2 -7049.741} C_VEL
LIN {X 0,Y 481.676,Z 290.482,A -85,B 0,C 180,E1 -7052.674,E2 -7052.674} C_VEL
LIN {X 0,Y 481.636,Z 290.488,A -85,B 0,C 180,E1 -7055.709,E2 -7055.709} C_VEL
LIN {X 0,Y 481.674,Z 290.482,A -85,B 0,C 180,E1 -7058.859,E2 -7058.859} C_VEL
LIN {X 0,Y 481.656,Z 290.485,A -85,B 0,C 180,E1 -7061.912,E2 -7061.912} C_VEL
LIN {X 0,Y 481.658,Z 290.482,A -85,B 0,C 180,E1 -7064.457,E2 -7064.457} C_VEL
LIN {X 0,Y 481.651,Z 290.49,A -85,B 0,C 180,E1 -7067.839,E2 -7067.839} C_VEL
LIN {X 0,Y 481.664,Z 290.481,A -85,B 0,C 180,E1 -7070.653,E2 -7070.653} C_VEL
LIN {X 0,Y 481.631,Z 290.488,A -85,B 0,C 180,E1 -7073.376,E2 -7073.376} C_VEL
LIN {X 0,Y 481.714,Z 290.479,A -85,B 0,C 180,E1 -7076.329,E2 -7076.329} C_VEL
LIN {X 0,Y 481.654,Z 290.484,A -85,B 0,C 180,E1 -7079.417,E2 -7079.417} C_VEL
LIN {X 0,Y 481.704,Z 290.485,A -85,B 0,C 180,E1 -7082.167,E2 -7082.167} C_VEL
LIN {X 0,Y 481.696,Z 290.478,A -85,B 0,C 180,E1 -7084.968,E2 -7084.968} C_VEL
LIN {X 0,Y 481.639,Z 290.485,A -85,B 0,C 180,E1 -7087.974,E2 -7087.974} C_VEL
LIN {X 0,Y 480.972,Z 290.573,A -85,B 0,C 180,E1 -7088.672,E2 -7088.672} C_VEL
LIN {X 0,Y 478.146,Z 290.921,A -85,B 0,C 180,E1 -7089.806,E2 -7089.806} C_VEL
LIN {X 0,Y 475.762,Z 291.221,A -85,B 0,C 180,E1 -7090.72,E2 -7090.72} C_VEL
LIN {X 0,Y 474.74,Z 291.344,A -85,B 0,C 180,E1 -7091.426,E2 -7091.426} C_VEL
LIN {X 0,Y 474.657,Z 291.354,A -85,B 0,C 180,E1 -7091.665,E2 -7091.665} C_VEL
LIN {X 0,Y 474.703,Z 291.358,A -85,B 0,C 180,E1 -7094.543,E2 -7094.543} C_VEL
LIN {X 0,Y 474.706,Z 291.349,A -85,B 0,C 180,E1 -7098.036,E2 -7098.036} C_VEL
LIN {X 0,Y 474.713,Z 291.351,A -85,B 0,C 180,E1 -7101.485,E2 -7101.485} C_VEL
LIN {X 0,Y 474.805,Z 291.424,A -85,B 0,C 180,E1 -7104.451,E2 -7104.451} C_VEL
LIN {X 0,Y 475.68,Z 297.726,A -85,B 0,C 180,E1 -7105.762,E2 -7105.762} C_VEL
LIN {X 0,Y 475.356,Z 310.685,A -85,B 0,C 180,E1 -7108.333,E2 -7108.333} C_VEL
LIN {X 0,Y 478.137,Z 325.41,A -85,B 0,C 180,E1 -7108.661,E2 -7108.661} C_VEL
LIN {X 0,Y 477.354,Z 417.95,A -85,B 0,C 180,E1 -7110.078,E2 -7110.078} C_VEL
LIN {X 0,Y 477.08,Z 431.033,A -85,B 0,C 180,E1 -7110.447,E2 -7110.447} C_VEL
LIN {X 0,Y 476.827,Z 444.101,A -85,B 0,C 180,E1 -7111.002,E2 -7111.002} C_VEL
LIN {X 0,Y 476.413,Z 455.969,A -85,B 0,C 180,E1 -7111.689,E2 -7111.689} C_VEL
LIN {X 0,Y 475.881,Z 467.363,A -85,B 0,C 180,E1 -7112.538,E2 -7112.538} C_VEL
LIN {X 0,Y 475.4,Z 477.633,A -85,B 0,C 180,E1 -7113.495,E2 -7113.495} C_VEL
LIN {X 0,Y 475.041,Z 486.027,A -85,B 0,C 180,E1 -7114.453,E2 -7114.453} C_VEL
LIN {X 0,Y 474.616,Z 495.148,A -85,B 0,C 180,E1 -7115.735,E2 -7115.735} C_VEL
LIN {X 0,Y 474.385,Z 502.251,A -85,B 0,C 180,E1 -7116.974,E2 -7116.974} C_VEL
LIN {X 0,Y 474.161,Z 507.494,A -85,B 0,C 180,E1 -7118.093,E2 -7118.093} C_VEL
LIN {X 0,Y 473.966,Z 512.357,A -85,B 0,C 180,E1 -7119.386,E2 -7119.386} C_VEL
LIN {X 0,Y 473.87,Z 516.095,A -85,B 0,C 180,E1 -7120.682,E2 -7120.682} C_VEL
LIN {X 0,Y 473.765,Z 518.808,A -85,B 0,C 180,E1 -7121.985,E2 -7121.985} C_VEL
LIN {X 0,Y 473.677,Z 520.088,A -85,B 0,C 180,E1 -7122.858,E2 -7122.858} C_VEL
LIN {X 0,Y 473.65,Z 520.943,A -85,B 0,C 180,E1 -7123.732,E2 -7123.732} C_VEL
LIN {X 0,Y 473.704,Z 521.379,A -85,B 0,C 180,E1 -7125.344,E2 -7125.344} C_VEL
LIN {X 0,Y 473.613,Z 520.959,A -85,B 0,C 180,E1 -7126.375,E2 -7126.375} C_VEL
LIN {X 0,Y 473.656,Z 520.096,A -85,B 0,C 180,E1 -7127.261,E2 -7127.261} C_VEL
LIN {X 0,Y 473.752,Z 518.542,A -85,B 0,C 180,E1 -7128.301,E2 -7128.301} C_VEL
LIN {X 0,Y 473.842,Z 515.984,A -85,B 0,C 180,E1 -7129.493,E2 -7129.493} C_VEL
LIN {X 0,Y 473.982,Z 511.816,A -85,B 0,C 180,E1 -7130.911,E2 -7130.911} C_VEL
LIN {X 0,Y 474.144,Z 506.811,A -85,B 0,C 180,E1 -7132.207,E2 -7132.207} C_VEL
LIN {X 0,Y 474.456,Z 500.101,A -85,B 0,C 180,E1 -7133.573,E2 -7133.573} C_VEL
LIN {X 0,Y 474.873,Z 491.547,A -85,B 0,C 180,E1 -7134.946,E2 -7134.946} C_VEL
LIN {X 0,Y 475.305,Z 482.643,A -85,B 0,C 180,E1 -7136.099,E2 -7136.099} C_VEL
LIN {X 0,Y 475.795,Z 472.755,A -85,B 0,C 180,E1 -7137.131,E2 -7137.131} C_VEL
LIN {X 0,Y 476.245,Z 461.26,A -85,B 0,C 180,E1 -7138.093,E2 -7138.093} C_VEL
LIN {X 0,Y 476.762,Z 449.454,A -85,B 0,C 180,E1 -7138.865,E2 -7138.865} C_VEL
LIN {X 0,Y 477.076,Z 438.25,A -85,B 0,C 180,E1 -7139.424,E2 -7139.424} C_VEL
LIN {X 0,Y 477.403,Z 424.883,A -85,B 0,C 180,E1 -7139.9,E2 -7139.9} C_VEL
LIN {X 0,Y 477.608,Z 412.701,A -85,B 0,C 180,E1 -7140.171,E2 -7140.171} C_VEL
LIN {X 0,Y 478.183,Z 324.321,A -85,B 0,C 180,E1 -7141.522,E2 -7141.522} C_VEL
LIN {X 0,Y 475.458,Z 310.587,A -85,B 0,C 180,E1 -7141.853,E2 -7141.853} C_VEL
LIN {X 0,Y 475.647,Z 297.278,A -85,B 0,C 180,E1 -7144.412,E2 -7144.412} C_VEL
LIN {X 0,Y 474.602,Z 291.37,A -85,B 0,C 180,E1 -7145.625,E2 -7145.625} C_VEL
LIN {X 0,Y 474.576,Z 291.37,A -85,B 0,C 180,E1 -7148.459,E2 -7148.459} C_VEL
LIN {X 0,Y 474.588,Z 291.368,A -85,B 0,C 180,E1 -7150.954,E2 -7150.954} C_VEL
LIN {X 0,Y 474.568,Z 291.368,A -85,B 0,C 180,E1 -7154.107,E2 -7154.107} C_VEL
LIN {X 0,Y 474.562,Z 291.367,A -85,B 0,C 180,E1 -7157.06,E2 -7157.06} C_VEL
LIN {X 0,Y 474.588,Z 291.365,A -85,B 0,C 180,E1 -7160.355,E2 -7160.355} C_VEL
LIN {X 0,Y 474.565,Z 291.366,A -85,B 0,C 180,E1 -7163.675,E2 -7163.675} C_VEL
LIN {X 0,Y 474.611,Z 291.362,A -85,B 0,C 180,E1 -7166.778,E2 -7166.778} C_VEL
LIN {X 0,Y 474.589,Z 291.371,A -85,B 0,C 180,E1 -7169.769,E2 -7169.769} C_VEL
LIN {X 0,Y 474.623,Z 291.36,A -85,B 0,C 180,E1 -7172.675,E2 -7172.675} C_VEL
LIN {X 0,Y 474.616,Z 291.361,A -85,B 0,C 180,E1 -7175.505,E2 -7175.505} C_VEL
LIN {X 0,Y 474.619,Z 291.356,A -85,B 0,C 180,E1 -7178.883,E2 -7178.883} C_VEL
LIN {X 0,Y 474.63,Z 291.365,A -85,B 0,C 180,E1 -7181.883,E2 -7181.883} C_VEL
LIN {X 0,Y 474.683,Z 291.355,A -85,B 0,C 180,E1 -7184.544,E2 -7184.544} C_VEL
LIN {X 0,Y 474.689,Z 291.353,A -85,B 0,C 180,E1 -7188.037,E2 -7188.037} C_VEL
LIN {X 0,Y 474.712,Z 291.348,A -85,B 0,C 180,E1 -7191.486,E2 -7191.486} C_VEL
LIN {X 0,Y 474.73,Z 291.348,A -85,B 0,C 180,E1 -7194.904,E2 -7194.904} C_VEL
LIN {X 0,Y 474.878,Z 291.324,A -85,B 0,C 180,E1 -7197.455,E2 -7197.455} C_VEL
LIN {X 0,Y 474.862,Z 291.333,A -85,B 0,C 180,E1 -7200.848,E2 -7200.848} C_VEL
LIN {X 0,Y 474.879,Z 291.329,A -85,B 0,C 180,E1 -7202.545,E2 -7202.545} C_VEL
LIN {X 0,Y 474.756,Z 291.343,A -85,B 0,C 180,E1 -7205.948,E2 -7205.948} C_VEL
LIN {X 0,Y 474.714,Z 291.349,A -85,B 0,C 180,E1 -7208.514,E2 -7208.514} C_VEL
LIN {X 0,Y 474.691,Z 291.35,A -85,B 0,C 180,E1 -7211.963,E2 -7211.963} C_VEL
LIN {X 0,Y 474.686,Z 291.353,A -85,B 0,C 180,E1 -7215.456,E2 -7215.456} C_VEL
LIN {X 0,Y 474.651,Z 291.358,A -85,B 0,C 180,E1 -7219.011,E2 -7219.011} C_VEL
LIN {X 0,Y 474.577,Z 291.365,A -85,B 0,C 180,E1 -7221.73,E2 -7221.73} C_VEL
LIN {X 0,Y 474.647,Z 291.354,A -85,B 0,C 180,E1 -7224.494,E2 -7224.494} C_VEL
LIN {X 0,Y 474.687,Z 291.353,A -85,B 0,C 180,E1 -7227.34,E2 -7227.34} C_VEL
LIN {X 0,Y 474.606,Z 291.365,A -85,B 0,C 180,E1 -7230.814,E2 -7230.814} C_VEL
LIN {X 0,Y 474.627,Z 291.361,A -85,B 0,C 180,E1 -7233.985,E2 -7233.985} C_VEL
LIN {X 0,Y 474.567,Z 291.368,A -85,B 0,C 180,E1 -7236.902,E2 -7236.902} C_VEL
LIN {X 0,Y 474.642,Z 291.364,A -85,B 0,C 180,E1 -7239.652,E2 -7239.652} C_VEL
LIN {X 0,Y 474.627,Z 291.36,A -85,B 0,C 180,E1 -7242.933,E2 -7242.933} C_VEL
LIN {X 0,Y 474.61,Z 291.36,A -85,B 0,C 180,E1 -7245.898,E2 -7245.898} C_VEL
LIN {X 0,Y 474.639,Z 291.359,A -85,B 0,C 180,E1 -7249.04,E2 -7249.04} C_VEL
LIN {X 0,Y 474.611,Z 291.369,A -85,B 0,C 180,E1 -7251.704,E2 -7251.704} C_VEL
LIN {X 0,Y 474.624,Z 291.362,A -85,B 0,C 180,E1 -7254.728,E2 -7254.728} C_VEL
LIN {X 0,Y 474.631,Z 291.367,A -85,B 0,C 180,E1 -7257.789,E2 -7257.789} C_VEL
LIN {X 0,Y 474.62,Z 291.363,A -85,B 0,C 180,E1 -7260.886,E2 -7260.886} C_VEL
LIN {X 0,Y 474.669,Z 291.359,A -85,B 0,C 180,E1 -7263.631,E2 -7263.631} C_VEL
LIN {X 0,Y 474.71,Z 291.487,A -85,B 0,C 180,E1 -7264.106,E2 -7264.106} C_VEL
LIN {X 0,Y 476.799,Z 302.761,A -85,B 0,C 180,E1 -7266.22,E2 -7266.22} C_VEL
LIN {X 0,Y 476.352,Z 315.838,A -85,B 0,C 180,E1 -7268.481,E2 -7268.481} C_VEL
LIN {X 0,Y 475.626,Z 334.779,A -85,B 0,C 180,E1 -7271.701,E2 -7271.701} C_VEL
LIN {X 0,Y 475.275,Z 343.64,A -85,B 0,C 180,E1 -7273.19,E2 -7273.19} C_VEL
LIN {X 0,Y 478.061,Z 361.636,A -85,B 0,C 180,E1 -7273.577,E2 -7273.577} C_VEL
LIN {X 0,Y 477.409,Z 452.954,A -85,B 0,C 180,E1 -7274.991,E2 -7274.991} C_VEL
LIN {X 0,Y 477.018,Z 466.681,A -85,B 0,C 180,E1 -7275.387,E2 -7275.387} C_VEL
LIN {X 0,Y 476.556,Z 479.028,A -85,B 0,C 180,E1 -7275.918,E2 -7275.918} C_VEL
LIN {X 0,Y 476.106,Z 491.677,A -85,B 0,C 180,E1 -7276.667,E2 -7276.667} C_VEL
LIN {X 0,Y 475.577,Z 502.794,A -85,B 0,C 180,E1 -7277.508,E2 -7277.508} C_VEL
LIN {X 0,Y 475.146,Z 513.096,A -85,B 0,C 180,E1 -7278.483,E2 -7278.483} C_VEL
LIN {X 0,Y 474.726,Z 522.259,A -85,B 0,C 180,E1 -7279.553,E2 -7279.553} C_VEL
LIN {X 0,Y 474.319,Z 531.197,A -85,B 0,C 180,E1 -7280.836,E2 -7280.836} C_VEL
LIN {X 0,Y 474.063,Z 538.397,A -85,B 0,C 180,E1 -7282.119,E2 -7282.119} C_VEL
LIN {X 0,Y 473.935,Z 543.265,A -85,B 0,C 180,E1 -7283.188,E2 -7283.188} C_VEL
LIN {X 0,Y 473.844,Z 548.002,A -85,B 0,C 180,E1 -7284.469,E2 -7284.469} C_VEL
LIN {X 0,Y 473.734,Z 551.62,A -85,B 0,C 180,E1 -7285.747,E2 -7285.747} C_VEL
LIN {X 0,Y 473.795,Z 553.49,A -85,B 0,C 180,E1 -7286.6,E2 -7286.6} C_VEL
LIN {X 0,Y 473.724,Z 555.889,A -85,B 0,C 180,E1 -7288.301,E2 -7288.301} C_VEL
LIN {X 0,Y 473.688,Z 556.499,A -85,B 0,C 180,E1 -7289.151,E2 -7289.151} C_VEL
LIN {X 0,Y 473.672,Z 556.714,A -85,B 0,C 180,E1 -7290.001,E2 -7290.001} C_VEL
LIN {X 0,Y 473.724,Z 555.889,A -85,B 0,C 180,E1 -7291.702,E2 -7291.702} C_VEL
LIN {X 0,Y 473.741,Z 554.89,A -85,B 0,C 180,E1 -7292.552,E2 -7292.552} C_VEL
LIN {X 0,Y 473.796,Z 553.488,A -85,B 0,C 180,E1 -7293.403,E2 -7293.403} C_VEL
LIN {X 0,Y 473.762,Z 550.537,A -85,B 0,C 180,E1 -7294.681,E2 -7294.681} C_VEL
LIN {X 0,Y 473.834,Z 546.543,A -85,B 0,C 180,E1 -7295.961,E2 -7295.961} C_VEL
LIN {X 0,Y 474.017,Z 540.397,A -85,B 0,C 180,E1 -7297.455,E2 -7297.455} C_VEL
LIN {X 0,Y 474.261,Z 533.686,A -85,B 0,C 180,E1 -7298.738,E2 -7298.738} C_VEL
LIN {X 0,Y 474.556,Z 525.351,A -85,B 0,C 180,E1 -7300.022,E2 -7300.022} C_VEL
LIN {X 0,Y 474.954,Z 516.787,A -85,B 0,C 180,E1 -7301.092,E2 -7301.092} C_VEL
LIN {X 0,Y 475.466,Z 506.446,A -85,B 0,C 180,E1 -7302.139,E2 -7302.139} C_VEL
LIN {X 0,Y 475.856,Z 496.016,A -85,B 0,C 180,E1 -7302.996,E2 -7302.996} C_VEL
LIN {X 0,Y 476.316,Z 484.202,A -85,B 0,C 180,E1 -7303.765,E2 -7303.765} C_VEL
LIN {X 0,Y 476.736,Z 472.26,A -85,B 0,C 180,E1 -7304.351,E2 -7304.351} C_VEL
LIN {X 0,Y 477.146,Z 459.374,A -85,B 0,C 180,E1 -7304.802,E2 -7304.802} C_VEL
LIN {X 0,Y 477.359,Z 445.829,A -85,B 0,C 180,E1 -7305.095,E2 -7305.095} C_VEL
LIN {X 0,Y 477.89,Z 361.313,A -85,B 0,C 180,E1 -7306.373,E2 -7306.373} C_VEL
LIN {X 0,Y 475.253,Z 343.88,A -85,B 0,C 180,E1 -7306.732,E2 -7306.732} C_VEL
LIN {X 0,Y 475.9,Z 326.772,A -85,B 0,C 180,E1 -7309.61,E2 -7309.61} C_VEL
LIN {X 0,Y 476.677,Z 306.846,A -85,B 0,C 180,E1 -7313,E2 -7313} C_VEL
LIN {X 0,Y 476.626,Z 301.639,A -85,B 0,C 180,E1 -7313.906,E2 -7313.906} C_VEL
LIN {X 0,Y 474.707,Z 291.357,A -85,B 0,C 180,E1 -7315.832,E2 -7315.832} C_VEL
LIN {X 0,Y 474.65,Z 291.363,A -85,B 0,C 180,E1 -7318.283,E2 -7318.283} C_VEL
LIN {X 0,Y 474.604,Z 291.361,A -85,B 0,C 180,E1 -7321.218,E2 -7321.218} C_VEL
LIN {X 0,Y 474.626,Z 291.367,A -85,B 0,C 180,E1 -7324.243,E2 -7324.243} C_VEL
LIN {X 0,Y 474.595,Z 291.362,A -85,B 0,C 180,E1 -7327.384,E2 -7327.384} C_VEL
LIN {X 0,Y 474.623,Z 291.365,A -85,B 0,C 180,E1 -7330.658,E2 -7330.658} C_VEL
LIN {X 0,Y 474.601,Z 291.361,A -85,B 0,C 180,E1 -7333.481,E2 -7333.481} C_VEL
LIN {X 0,Y 474.606,Z 291.367,A -85,B 0,C 180,E1 -7336.519,E2 -7336.519} C_VEL
LIN {X 0,Y 474.623,Z 291.36,A -85,B 0,C 180,E1 -7339.343,E2 -7339.343} C_VEL
LIN {X 0,Y 474.595,Z 291.367,A -85,B 0,C 180,E1 -7342.616,E2 -7342.616} C_VEL
LIN {X 0,Y 474.625,Z 291.358,A -85,B 0,C 180,E1 -7345.758,E2 -7345.758} C_VEL
LIN {X 0,Y 474.604,Z 291.365,A -85,B 0,C 180,E1 -7348.782,E2 -7348.782} C_VEL
LIN {X 0,Y 474.651,Z 291.357,A -85,B 0,C 180,E1 -7351.718,E2 -7351.718} C_VEL
LIN {X 0,Y 474.659,Z 291.355,A -85,B 0,C 180,E1 -7354.582,E2 -7354.582} C_VEL
LIN {X 0,Y 474.607,Z 291.37,A -85,B 0,C 180,E1 -7357.355,E2 -7357.355} C_VEL
LIN {X 0,Y 474.66,Z 291.355,A -85,B 0,C 180,E1 -7360.09,E2 -7360.09} C_VEL
LIN {X 0,Y 474.643,Z 291.356,A -85,B 0,C 180,E1 -7362.774,E2 -7362.774} C_VEL
LIN {X 0,Y 474.653,Z 291.361,A -85,B 0,C 180,E1 -7365.421,E2 -7365.421} C_VEL
LIN {X 0,Y 474.71,Z 291.352,A -85,B 0,C 180,E1 -7368.038,E2 -7368.038} C_VEL
LIN {X 0,Y 474.731,Z 291.349,A -85,B 0,C 180,E1 -7371.486,E2 -7371.486} C_VEL
LIN {X 0,Y 474.75,Z 291.342,A -85,B 0,C 180,E1 -7374.904,E2 -7374.904} C_VEL
LIN {X 0,Y 474.898,Z 291.326,A -85,B 0,C 180,E1 -7377.455,E2 -7377.455} C_VEL
LIN {X 0,Y 474.915,Z 291.33,A -85,B 0,C 180,E1 -7380,E2 -7380} C_VEL
LIN {X 0,Y 474.897,Z 291.328,A -85,B 0,C 180,E1 -7382.544,E2 -7382.544} C_VEL
LIN {X 0,Y 474.773,Z 291.344,A -85,B 0,C 180,E1 -7385.947,E2 -7385.947} C_VEL
LIN {X 0,Y 474.716,Z 291.354,A -85,B 0,C 180,E1 -7388.514,E2 -7388.514} C_VEL
LIN {X 0,Y 474.709,Z 291.35,A -85,B 0,C 180,E1 -7391.962,E2 -7391.962} C_VEL
LIN {X 0,Y 474.705,Z 291.348,A -85,B 0,C 180,E1 -7395.455,E2 -7395.455} C_VEL
LIN {X 0,Y 474.667,Z 291.358,A -85,B 0,C 180,E1 -7399.01,E2 -7399.01} C_VEL
LIN {X 0,Y 474.593,Z 291.362,A -85,B 0,C 180,E1 -7401.729,E2 -7401.729} C_VEL
LIN {X 0,Y 474.661,Z 291.357,A -85,B 0,C 180,E1 -7404.493,E2 -7404.493} C_VEL
